C07331=1159.961,302.265,-72.493,-176.878,8.230,148.701
C07332=1159.957,302.514,-72.524,-176.876,8.233,148.700
C07333=1159.952,302.762,-72.555,-176.873,8.237,148.701
C07334=1159.948,303.010,-72.586,-176.871,8.239,148.701
C07335=1159.944,303.258,-72.616,-176.868,8.243,148.701
C07336=1159.940,303.506,-72.648,-176.866,8.246,148.701
C07337=1159.936,303.754,-72.679,-176.863,8.249,148.701
C07338=1159.932,304.002,-72.710,-176.861,8.252,148.701
C07339=1159.928,304.250,-72.740,-176.858,8.256,148.701
C07340=1159.923,304.498,-72.771,-176.855,8.259,148.701
C07341=1159.919,304.747,-72.802,-176.853,8.262,148.701
C07342=1159.914,304.994,-72.833,-176.850,8.265,148.701
C07343=1159.910,305.242,-72.863,-176.848,8.269,148.701
C07344=1159.906,305.490,-72.895,-176.845,8.272,148.701
C07345=1159.902,305.738,-72.925,-176.842,8.275,148.702
C07346=1159.898,305.986,-72.956,-176.840,8.278,148.702
C07347=1159.894,306.235,-72.987,-176.837,8.282,148.702
C07348=1159.889,306.482,-73.019,-176.835,8.285,148.702
C07349=1159.885,306.731,-73.050,-176.832,8.288,148.702
C07350=1159.881,306.979,-73.081,-176.830,8.291,148.702
C07351=1159.876,307.227,-73.111,-176.827,8.294,148.702
C07352=1159.873,307.474,-73.143,-176.824,8.298,148.702
C07353=1159.868,307.722,-73.173,-176.822,8.301,148.702
C07354=1159.864,307.971,-73.205,-176.819,8.305,148.703
C07355=1159.860,308.218,-73.236,-176.816,8.308,148.703
C07356=1159.856,308.466,-73.267,-176.814,8.311,148.703
C07357=1159.852,308.715,-73.298,-176.811,8.314,148.703
C07358=1159.847,308.962,-73.329,-176.809,8.317,148.703
C07359=1159.843,309.211,-73.361,-176.806,8.320,148.703
C07360=1159.839,309.458,-73.392,-176.804,8.323,148.703
C07361=1159.835,309.707,-73.423,-176.801,8.328,148.703
C07362=1159.830,309.955,-73.454,-176.798,8.331,148.703
C07363=1159.827,310.203,-73.486,-176.796,8.334,148.703
C07364=1159.822,310.451,-73.517,-176.793,8.337,148.704
C07365=1159.818,310.699,-73.548,-176.791,8.340,148.704
C07366=1159.814,310.947,-73.579,-176.788,8.343,148.704
C07367=1159.810,311.195,-73.611,-176.785,8.347,148.704
C07368=1159.805,311.443,-73.642,-176.783,8.350,148.704
C07369=1159.802,311.691,-73.674,-176.780,8.354,148.704
C07370=1159.797,311.939,-73.704,-176.778,8.357,148.704
C07371=1159.793,312.187,-73.736,-176.775,8.360,148.704
C07372=1159.789,312.434,-73.768,-176.773,8.363,148.705
C07373=1159.785,312.683,-73.799,-176.770,8.367,148.705
C07374=1159.781,312.930,-73.830,-176.767,8.370,148.705
C07375=1159.777,313.179,-73.861,-176.765,8.373,148.705
C07376=1159.772,313.456,-73.897,-176.762,8.377,148.705
C07377=1159.767,313.733,-73.932,-176.760,8.381,148.705
C07378=1159.762,314.010,-73.967,-176.756,8.384,148.705
C07379=1159.758,314.288,-74.003,-176.753,8.389,148.705
C07380=1159.754,314.536,-74.034,-176.751,8.392,148.705
C07381=1159.750,314.784,-74.066,-176.748,8.395,148.706
C07382=1159.745,315.031,-74.098,-176.746,8.398,148.706
C07383=1159.741,315.280,-74.129,-176.743,8.401,148.706
C07384=1159.737,315.528,-74.161,-176.741,8.404,148.706
C07385=1159.733,315.775,-74.192,-176.738,8.408,148.706
C07386=1159.729,316.023,-74.224,-176.735,8.411,148.706
C07387=1159.724,316.271,-74.256,-176.733,8.415,148.706
C07388=1159.720,316.520,-74.287,-176.731,8.418,148.707
C07389=1159.716,316.768,-74.319,-176.728,8.421,148.707
C07390=1159.712,317.015,-74.351,-176.725,8.425,148.707
C07391=1159.708,317.263,-74.382,-176.723,8.428,148.707
C07392=1159.703,317.511,-74.415,-176.720,8.431,148.707
C07393=1159.700,317.759,-74.446,-176.718,8.435,148.707
C07394=1159.696,318.007,-74.478,-176.715,8.438,148.707
C07395=1159.691,318.255,-74.509,-176.712,8.442,148.707
C07396=1159.687,318.503,-74.541,-176.710,8.445,148.708
C07397=1159.683,318.751,-74.573,-176.707,8.448,148.708
C07398=1159.679,318.998,-74.605,-176.705,8.451,148.708
C07399=1159.674,319.247,-74.637,-176.702,8.454,148.708
C07400=1159.671,319.495,-74.669,-176.699,8.459,148.708
C07401=1159.666,319.742,-74.701,-176.697,8.462,148.708
C07402=1159.663,319.990,-74.732,-176.694,8.465,148.708
C07403=1159.658,320.239,-74.765,-176.692,8.468,148.709
C07404=1159.654,320.487,-74.797,-176.689,8.472,148.709
C07405=1159.650,320.734,-74.828,-176.687,8.475,148.709
C07406=1159.646,320.982,-74.861,-176.684,8.478,148.709
C07407=1159.642,321.230,-74.892,-176.682,8.482,148.709
C07408=1159.637,321.478,-74.924,-176.680,8.485,148.709
C07409=1159.634,321.725,-74.957,-176.677,8.489,148.710
C07410=1159.630,321.973,-74.989,-176.674,8.492,148.710
C07411=1159.625,322.222,-75.021,-176.672,8.495,148.710
C07412=1159.621,322.469,-75.053,-176.669,8.499,148.710
C07413=1159.617,322.717,-75.085,-176.666,8.502,148.710
C07414=1159.613,322.966,-75.117,-176.664,8.506,148.710
C07415=1159.609,323.214,-75.149,-176.661,8.509,148.710
C07416=1159.604,323.461,-75.182,-176.659,8.512,148.711
C07417=1159.601,323.709,-75.214,-176.657,8.516,148.711
C07418=1159.596,323.957,-75.246,-176.653,8.519,148.711
C07419=1159.593,324.205,-75.278,-176.651,8.523,148.711
C07420=1159.588,324.453,-75.311,-176.649,8.526,148.711
C07421=1159.584,324.700,-75.342,-176.647,8.529,148.711
C07422=1159.580,324.948,-75.375,-176.643,8.533,148.711
C07423=1159.576,325.196,-75.407,-176.641,8.536,148.712
C07424=1159.572,325.444,-75.440,-176.639,8.540,148.712
C07425=1159.568,325.692,-75.472,-176.636,8.543,148.712
C07426=1159.563,325.940,-75.504,-176.633,8.547,148.712
C07427=1159.560,326.187,-75.536,-176.631,8.550,148.712
C07428=1159.555,326.436,-75.569,-176.628,8.553,148.712
C07429=1159.552,326.684,-75.601,-176.626,8.557,148.713
C07430=1159.547,326.931,-75.634,-176.623,8.561,148.713
C07431=1159.542,327.179,-75.666,-176.621,8.564,148.713
C07432=1159.539,327.426,-75.698,-176.618,8.567,148.713
C07433=1159.535,327.675,-75.731,-176.616,8.570,148.713
C07434=1159.531,327.922,-75.763,-176.613,8.574,148.713
C07435=1159.527,328.171,-75.796,-176.611,8.578,148.714
C07436=1159.522,328.419,-75.828,-176.608,8.581,148.714
C07437=1159.519,328.666,-75.861,-176.605,8.585,148.714
C07438=1159.514,328.914,-75.893,-176.603,8.588,148.714
C07439=1159.510,329.162,-75.926,-176.600,8.591,148.714
C07440=1159.506,329.409,-75.959,-176.598,8.594,148.715
C07441=1159.502,329.658,-75.991,-176.595,8.599,148.715
C07442=1159.498,329.905,-76.024,-176.593,8.602,148.715
C07443=1159.494,330.153,-76.056,-176.591,8.605,148.715
C07444=1159.490,330.401,-76.089,-176.588,8.608,148.715
C07445=1159.485,330.649,-76.122,-176.585,8.612,148.715
C07446=1159.482,330.897,-76.154,-176.583,8.615,148.716
C07447=1159.478,331.145,-76.187,-176.580,8.619,148.716
C07448=1159.473,331.393,-76.220,-176.578,8.623,148.716
C07449=1159.469,331.640,-76.253,-176.575,8.626,148.716
C07450=1159.465,331.887,-76.285,-176.573,8.629,148.716
C07451=1159.461,332.136,-76.318,-176.571,8.633,148.717
C07452=1159.457,332.383,-76.351,-176.567,8.637,148.717
C07453=1159.453,332.631,-76.384,-176.565,8.640,148.717
C07454=1159.448,332.879,-76.416,-176.563,8.643,148.717
C07455=1159.445,333.127,-76.449,-176.560,8.647,148.717
C07456=1159.441,333.375,-76.482,-176.557,8.650,148.718
C07457=1159.436,333.622,-76.515,-176.555,8.654,148.718
C07458=1159.432,333.871,-76.548,-176.553,8.657,148.718
C07459=1159.428,334.118,-76.581,-176.550,8.661,148.718
C07460=1159.424,334.366,-76.613,-176.548,8.664,148.718
C07461=1159.420,334.614,-76.647,-176.545,8.668,148.719
C07462=1159.416,334.861,-76.680,-176.543,8.672,148.719
C07463=1159.412,335.109,-76.713,-176.540,8.675,148.719
C07464=1159.408,335.357,-76.745,-176.537,8.678,148.719
C07465=1159.403,335.605,-76.779,-176.535,8.682,148.719
C07466=1159.399,335.853,-76.812,-176.532,8.685,148.719
C07467=1159.395,336.101,-76.845,-176.530,8.689,148.720
C07468=1159.392,336.348,-76.877,-176.527,8.693,148.720
C07469=1159.388,336.596,-76.911,-176.525,8.696,148.720
C07470=1159.384,336.843,-76.944,-176.522,8.699,148.720
C07471=1159.379,337.091,-76.977,-176.520,8.704,148.721
C07472=1159.375,337.339,-77.010,-176.517,8.707,148.721
C07473=1159.372,337.587,-77.044,-176.515,8.710,148.721
C07474=1159.368,337.835,-77.077,-176.512,8.714,148.721
C07475=1159.363,338.083,-77.110,-176.510,8.717,148.721
C07476=1159.359,338.331,-77.143,-176.507,8.721,148.722
C07477=1159.355,338.578,-77.176,-176.505,8.725,148.722
C07478=1159.351,338.826,-77.209,-176.502,8.728,148.722
C07479=1159.347,339.074,-77.243,-176.500,8.731,148.722
C07480=1159.342,339.353,-77.280,-176.497,8.736,148.723
C07481=1159.338,339.633,-77.318,-176.494,8.740,148.723
C07482=1159.334,339.913,-77.355,-176.491,8.744,148.723
C07483=1159.329,340.193,-77.393,-176.488,8.748,148.723
C07484=1159.324,340.441,-77.427,-176.486,8.751,148.724
C07485=1159.320,340.689,-77.460,-176.483,8.755,148.724
C07486=1159.316,340.936,-77.493,-176.481,8.759,148.724
C07487=1159.312,341.183,-77.527,-176.479,8.762,148.724
C07488=1159.308,341.431,-77.560,-176.476,8.766,148.724
C07489=1159.304,341.679,-77.593,-176.473,8.769,148.725
C07490=1159.300,341.927,-77.627,-176.471,8.772,148.725
C07491=1159.296,342.174,-77.661,-176.468,8.777,148.725
C07492=1159.292,342.422,-77.694,-176.466,8.780,148.725
C07493=1159.287,342.670,-77.728,-176.464,8.783,148.726
C07494=1159.283,342.918,-77.761,-176.461,8.787,148.726
C07495=1159.279,343.165,-77.795,-176.458,8.791,148.726
C07496=1159.276,343.413,-77.828,-176.456,8.794,148.726
C07497=1159.272,343.661,-77.861,-176.453,8.798,148.726
C07498=1159.268,343.908,-77.895,-176.451,8.801,148.727
C07499=1159.263,344.156,-77.929,-176.449,8.806,148.727
C07500=1159.259,344.404,-77.962,-176.446,8.809,148.727
C07501=1159.256,344.652,-77.996,-176.444,8.812,148.728
C07502=1159.252,344.900,-78.029,-176.441,8.816,148.728
C07503=1159.247,345.147,-78.064,-176.439,8.820,148.728
C07504=1159.243,345.395,-78.097,-176.436,8.823,148.728
C07505=1159.239,345.642,-78.131,-176.434,8.827,148.728
C07506=1159.236,345.890,-78.164,-176.431,8.830,148.729
C07507=1159.231,346.138,-78.199,-176.428,8.834,148.729
C07508=1159.227,346.385,-78.232,-176.426,8.838,148.729
C07509=1159.223,346.632,-78.266,-176.424,8.841,148.729
C07510=1159.219,346.881,-78.299,-176.421,8.845,148.730
C07511=1159.215,347.128,-78.334,-176.419,8.849,148.730
C07512=1159.211,347.376,-78.367,-176.416,8.853,148.730
C07513=1159.208,347.624,-78.401,-176.414,8.856,148.730
C07514=1159.203,347.872,-78.435,-176.411,8.859,148.731
C07515=1159.199,348.119,-78.469,-176.409,8.863,148.731
C07516=1159.195,348.366,-78.503,-176.406,8.867,148.731
C07517=1159.191,348.615,-78.537,-176.404,8.871,148.732
C07518=1159.187,348.862,-78.571,-176.402,8.874,148.732
C07519=1159.183,349.110,-78.604,-176.399,8.878,148.732
C07520=1159.179,349.358,-78.639,-176.396,8.882,148.732
C07521=1159.175,349.605,-78.673,-176.394,8.885,148.733
C07522=1159.170,349.853,-78.706,-176.391,8.889,148.733
C07523=1159.167,350.101,-78.741,-176.389,8.892,148.733
C07524=1159.163,350.348,-78.775,-176.386,8.897,148.733
C07525=1159.158,350.595,-78.809,-176.384,8.900,148.734
C07526=1159.155,350.844,-78.843,-176.382,8.903,148.734
C07527=1159.150,351.091,-78.877,-176.379,8.908,148.734
C07528=1159.146,351.338,-78.911,-176.377,8.911,148.734
C07529=1159.143,351.586,-78.946,-176.374,8.915,148.735
C07530=1159.139,351.834,-78.980,-176.372,8.919,148.735
C07531=1159.134,352.082,-79.013,-176.369,8.923,148.735
C07532=1159.131,352.329,-79.048,-176.367,8.926,148.736
C07533=1159.126,352.577,-79.082,-176.364,8.929,148.736
C07534=1159.123,352.825,-79.116,-176.362,8.934,148.736
C07535=1159.118,353.072,-79.151,-176.360,8.937,148.736
C07536=1159.114,353.319,-79.185,-176.357,8.941,148.737
C07537=1159.110,353.567,-79.219,-176.354,8.944,148.737
C07538=1159.107,353.814,-79.253,-176.352,8.949,148.737
C07539=1159.103,354.062,-79.288,-176.350,8.952,148.738
C07540=1159.099,354.310,-79.322,-176.347,8.956,148.738
C07541=1159.094,354.557,-79.356,-176.344,8.959,148.738
C07542=1159.091,354.805,-79.390,-176.343,8.963,148.738
C07543=1159.086,355.053,-79.424,-176.340,8.967,148.739
C07544=1159.083,355.300,-79.459,-176.337,8.970,148.739
C07545=1159.079,355.547,-79.494,-176.335,8.974,148.739
C07546=1159.075,355.796,-79.529,-176.333,8.978,148.740
C07547=1159.071,356.043,-79.563,-176.330,8.982,148.740
C07548=1159.067,356.291,-79.597,-176.327,8.985,148.740
C07549=1159.062,356.538,-79.632,-176.325,8.990,148.741
C07550=1159.059,356.786,-79.666,-176.323,8.993,148.741
C07551=1159.054,357.033,-79.701,-176.320,8.997,148.741
C07552=1159.051,357.281,-79.735,-176.317,9.001,148.741
C07553=1159.047,357.529,-79.769,-176.315,9.005,148.742
C07554=1159.043,357.777,-79.804,-176.313,9.008,148.742
C07555=1159.039,358.023,-79.839,-176.310,9.012,148.742
C07556=1159.035,358.271,-79.874,-176.308,9.016,148.743
C07557=1159.031,358.519,-79.908,-176.305,9.020,148.743
C07558=1159.027,358.767,-79.943,-176.303,9.023,148.743
C07559=1159.023,359.013,-79.977,-176.300,9.028,148.744
C07560=1159.019,359.262,-80.012,-176.298,9.031,148.744
C07561=1159.015,359.509,-80.047,-176.295,9.035,148.744
C07562=1159.011,359.757,-80.081,-176.293,9.039,148.744
C07563=1159.007,360.004,-80.116,-176.290,9.043,148.745
C07564=1159.003,360.252,-80.151,-176.288,9.046,148.745
C07565=1158.999,360.499,-80.185,-176.286,9.051,148.745
C07566=1158.996,360.746,-80.220,-176.283,9.054,148.746
C07567=1158.992,360.994,-80.255,-176.280,9.058,148.746
C07568=1158.987,361.242,-80.290,-176.279,9.062,148.746
C07569=1158.983,361.489,-80.325,-176.276,9.066,148.747
C07570=1158.979,361.737,-80.360,-176.273,9.070,148.747
C07571=1158.976,361.985,-80.394,-176.271,9.073,148.747
C07572=1158.972,362.232,-80.429,-176.268,9.077,148.748
C07573=1158.967,362.480,-80.464,-176.266,9.081,148.748
C07574=1158.964,362.727,-80.499,-176.263,9.085,148.748
C07575=1158.959,362.974,-80.534,-176.261,9.089,148.749
C07576=1158.955,363.222,-80.569,-176.258,9.093,148.749
C07577=1158.952,363.470,-80.604,-176.256,9.097,148.749
C07578=1158.948,363.717,-80.639,-176.254,9.101,148.750
C07579=1158.944,363.965,-80.674,-176.251,9.105,148.750
C07580=1158.940,364.212,-80.709,-176.249,9.108,148.750
C07581=1158.936,364.460,-80.744,-176.246,9.112,148.751
C07582=1158.932,364.707,-80.779,-176.244,9.116,148.751
C07583=1158.928,364.955,-80.815,-176.241,9.120,148.751
C07584=1158.924,365.238,-80.854,-176.239,9.124,148.752
C07585=1158.919,365.520,-80.894,-176.236,9.129,148.752
C07586=1158.915,365.803,-80.934,-176.234,9.133,148.752
C07587=1158.910,366.086,-80.975,-176.230,9.138,148.753
C07588=1158.906,366.333,-81.010,-176.229,9.142,148.753
C07589=1158.902,366.580,-81.046,-176.226,9.146,148.754
C07590=1158.898,366.828,-81.081,-176.224,9.149,148.754
C07591=1158.894,367.075,-81.116,-176.221,9.154,148.755
C07592=1158.890,367.323,-81.151,-176.220,9.157,148.755
C07593=1158.886,367.571,-81.186,-176.217,9.162,148.755
C07594=1158.883,367.818,-81.222,-176.215,9.165,148.756
C07595=1158.878,368.065,-81.257,-176.212,9.170,148.756
C07596=1158.875,368.313,-81.292,-176.210,9.173,148.757
C07597=1158.871,368.560,-81.328,-176.208,9.177,148.757
C07598=1158.867,368.808,-81.362,-176.206,9.181,148.757
C07599=1158.863,369.055,-81.398,-176.203,9.185,148.758
C07600=1158.859,369.303,-81.433,-176.201,9.189,148.758
C07601=1158.856,369.550,-81.469,-176.199,9.193,148.759
C07602=1158.851,369.797,-81.504,-176.197,9.197,148.759
C07603=1158.848,370.044,-81.540,-176.195,9.201,148.760
C07604=1158.843,370.292,-81.576,-176.193,9.205,148.760
C07605=1158.839,370.540,-81.611,-176.191,9.208,148.760
C07606=1158.836,370.788,-81.646,-176.188,9.213,148.761
C07607=1158.831,371.035,-81.681,-176.186,9.216,148.761
C07608=1158.828,371.282,-81.717,-176.184,9.221,148.762
C07609=1158.824,371.530,-81.753,-176.182,9.224,148.762
C07610=1158.820,371.777,-81.788,-176.180,9.228,148.763
C07611=1158.816,372.025,-81.824,-176.178,9.233,148.763
C07612=1158.812,372.272,-81.859,-176.176,9.236,148.764
C07613=1158.808,372.519,-81.895,-176.174,9.241,148.764
C07614=1158.804,372.767,-81.931,-176.172,9.244,148.765
C07615=1158.801,373.014,-81.966,-176.171,9.248,148.765
C07616=1158.796,373.262,-82.002,-176.169,9.252,148.766
C07617=1158.793,373.509,-82.038,-176.166,9.256,148.766
C07618=1158.788,373.756,-82.073,-176.165,9.260,148.767
C07619=1158.785,374.003,-82.109,-176.163,9.264,148.767
C07620=1158.781,374.251,-82.145,-176.161,9.268,148.768
C07621=1158.777,374.498,-82.181,-176.159,9.272,148.768
C07622=1158.773,374.746,-82.216,-176.158,9.276,148.769
C07623=1158.770,374.993,-82.252,-176.156,9.280,148.769
C07624=1158.765,375.241,-82.288,-176.154,9.283,148.770
C07625=1158.761,375.488,-82.323,-176.153,9.287,148.771
C07626=1158.758,375.735,-82.360,-176.150,9.292,148.771
C07627=1158.753,375.983,-82.396,-176.149,9.296,148.772
C07628=1158.750,376.230,-82.431,-176.147,9.300,148.772
C07629=1158.746,376.478,-82.467,-176.146,9.303,148.773
C07630=1158.742,376.725,-82.502,-176.144,9.307,148.774
C07631=1158.738,376.972,-82.539,-176.143,9.311,148.774
C07632=1158.734,377.220,-82.575,-176.141,9.315,148.775
C07633=1158.731,377.467,-82.610,-176.140,9.319,148.775
C07634=1158.726,377.715,-82.646,-176.138,9.323,148.776
C07635=1158.722,377.961,-82.682,-176.137,9.327,148.776
C07636=1158.718,378.209,-82.719,-176.135,9.330,148.777
C07637=1158.714,378.457,-82.754,-176.134,9.334,148.778
C07638=1158.711,378.704,-82.790,-176.133,9.339,148.779
C07639=1158.707,378.951,-82.826,-176.131,9.342,148.779
C07640=1158.703,379.199,-82.862,-176.131,9.346,148.780
C07641=1158.699,379.446,-82.899,-176.129,9.349,148.780
C07642=1158.695,379.694,-82.934,-176.128,9.354,148.781
C07643=1158.692,379.941,-82.970,-176.127,9.358,148.782
C07644=1158.687,380.188,-83.007,-176.126,9.361,148.782
C07645=1158.684,380.436,-83.042,-176.125,9.365,148.783
C07646=1158.680,380.683,-83.079,-176.123,9.369,148.784
C07647=1158.676,380.931,-83.115,-176.123,9.372,148.785
C07648=1158.672,381.178,-83.151,-176.121,9.376,148.785
C07649=1158.668,381.425,-83.187,-176.120,9.380,148.786
C07650=1158.665,381.673,-83.223,-176.119,9.383,148.787
C07651=1158.661,381.920,-83.260,-176.118,9.388,148.787
C07652=1158.656,382.167,-83.295,-176.118,9.391,148.788
C07653=1158.652,382.414,-83.332,-176.117,9.395,148.789
C07654=1158.649,382.661,-83.367,-176.116,9.398,148.790
C07655=1158.644,382.909,-83.404,-176.116,9.402,148.790
C07656=1158.641,383.156,-83.440,-176.114,9.405,148.791
C07657=1158.637,383.403,-83.476,-176.114,9.409,148.792
C07658=1158.633,383.651,-83.512,-176.113,9.412,148.793
C07659=1158.629,383.898,-83.549,-176.112,9.416,148.793
C07660=1158.625,384.145,-83.584,-176.112,9.420,148.794
C07661=1158.621,384.393,-83.621,-176.111,9.423,148.795
C07662=1158.617,384.640,-83.657,-176.111,9.427,148.796
C07663=1158.613,384.887,-83.694,-176.110,9.430,148.796
C07664=1158.610,385.136,-83.730,-176.110,9.433,148.797
C07665=1158.606,385.383,-83.766,-176.110,9.437,148.798
C07666=1158.602,385.630,-83.803,-176.109,9.440,148.799
C07667=1158.598,385.877,-83.839,-176.109,9.444,148.800
C07668=1158.594,386.125,-83.876,-176.109,9.447,148.800
C07669=1158.591,386.372,-83.911,-176.109,9.450,148.801
C07670=1158.587,386.619,-83.948,-176.108,9.453,148.802
C07671=1158.583,386.866,-83.984,-176.108,9.457,148.803
C07672=1158.579,387.114,-84.021,-176.108,9.460,148.804
C07673=1158.576,387.361,-84.057,-176.108,9.463,148.804
C07674=1158.571,387.608,-84.094,-176.108,9.467,148.805
C07675=1158.567,387.856,-84.130,-176.108,9.469,148.806
C07676=1158.564,388.103,-84.166,-176.108,9.472,148.807
C07677=1158.560,388.350,-84.203,-176.108,9.475,148.808
C07678=1158.556,388.597,-84.238,-176.108,9.479,148.808
C07679=1158.552,388.845,-84.275,-176.108,9.482,148.809
C07680=1158.548,389.092,-84.312,-176.108,9.484,148.810
C07681=1158.544,389.339,-84.348,-176.108,9.488,148.811
C07682=1158.540,389.587,-84.385,-176.109,9.490,148.812
C07683=1158.537,389.833,-84.421,-176.109,9.493,148.813
C07684=1158.532,390.081,-84.457,-176.109,9.497,148.813
C07685=1158.529,390.328,-84.493,-176.109,9.500,148.814
C07686=1158.525,390.576,-84.530,-176.109,9.502,148.815
C07687=1158.521,390.824,-84.567,-176.110,9.505,148.816
C07688=1158.517,391.109,-84.609,-176.110,9.508,148.817
C07689=1158.512,391.395,-84.651,-176.110,9.512,148.818
C07690=1158.508,391.680,-84.693,-176.111,9.514,148.819
C07691=1158.503,391.966,-84.735,-176.112,9.517,148.820
C07692=1158.500,392.214,-84.772,-176.112,9.520,148.820
C07693=1158.496,392.461,-84.808,-176.112,9.523,148.821
C07694=1158.492,392.709,-84.844,-176.113,9.526,148.822
C07695=1158.488,392.956,-84.881,-176.113,9.529,148.823
C07696=1158.484,393.203,-84.918,-176.113,9.531,148.824
C07697=1158.480,393.451,-84.954,-176.114,9.534,148.825
C07698=1158.477,393.698,-84.990,-176.115,9.536,148.825
C07699=1158.472,393.945,-85.027,-176.115,9.539,148.826
C07700=1158.468,394.192,-85.064,-176.116,9.541,148.827
C07701=1158.465,394.439,-85.099,-176.116,9.543,148.828
C07702=1158.461,394.687,-85.136,-176.117,9.546,148.829
C07703=1158.457,394.934,-85.173,-176.117,9.549,148.829
C07704=1158.454,395.181,-85.210,-176.118,9.551,148.830
C07705=1158.450,395.429,-85.246,-176.119,9.554,148.831
C07706=1158.445,395.676,-85.283,-176.119,9.556,148.832
C07707=1158.442,395.923,-85.319,-176.120,9.558,148.833
C07708=1158.438,396.170,-85.356,-176.120,9.561,148.833
C07709=1158.434,396.418,-85.393,-176.121,9.563,148.834
C07710=1158.430,396.665,-85.428,-176.122,9.566,148.835
C07711=1158.426,396.912,-85.465,-176.123,9.567,148.836
C07712=1158.422,397.159,-85.502,-176.123,9.570,148.837
C07713=1158.419,397.406,-85.538,-176.124,9.572,148.837
C07714=1158.414,397.654,-85.575,-176.124,9.575,148.838
C07715=1158.410,397.901,-85.611,-176.125,9.577,148.839
C07716=1158.407,398.149,-85.648,-176.126,9.579,148.840
C07717=1158.403,398.396,-85.685,-176.126,9.581,148.840
C07718=1158.399,398.643,-85.721,-176.127,9.583,148.841
C07719=1158.395,398.891,-85.757,-176.128,9.586,148.842
C07720=1158.391,399.138,-85.794,-176.129,9.588,148.843
C07721=1158.387,399.385,-85.831,-176.129,9.590,148.843
C07722=1158.384,399.632,-85.867,-176.131,9.592,148.844
C07723=1158.380,399.879,-85.904,-176.131,9.594,148.845
C07724=1158.375,400.127,-85.940,-176.132,9.596,148.846
C07725=1158.372,400.374,-85.976,-176.132,9.598,148.846
C07726=1158.369,400.622,-86.013,-176.133,9.601,148.847
C07727=1158.364,400.869,-86.050,-176.134,9.603,148.848
C07728=1158.361,401.116,-86.087,-176.134,9.605,148.849
C07729=1158.357,401.364,-86.123,-176.136,9.607,148.849
C07730=1158.353,401.611,-86.160,-176.136,9.608,148.850
C07731=1158.349,401.858,-86.196,-176.137,9.611,148.851
C07732=1158.345,402.105,-86.233,-176.137,9.613,148.852
C07733=1158.341,402.352,-86.270,-176.138,9.615,148.852
C07734=1158.337,402.599,-86.306,-176.139,9.617,148.853
C07735=1158.333,402.847,-86.342,-176.140,9.619,148.854
C07736=1158.330,403.095,-86.379,-176.140,9.621,148.854
C07737=1158.326,403.342,-86.416,-176.141,9.623,148.855
C07738=1158.322,403.589,-86.452,-176.142,9.625,148.856
C07739=1158.318,403.836,-86.489,-176.143,9.627,148.857
C07740=1158.314,404.084,-86.525,-176.143,9.628,148.857
C07741=1158.310,404.331,-86.562,-176.144,9.630,148.858
C07742=1158.306,404.578,-86.598,-176.145,9.632,148.859
C07743=1158.302,404.825,-86.635,-176.145,9.635,148.859
C07744=1158.299,405.072,-86.672,-176.146,9.637,148.860
C07745=1158.295,405.320,-86.709,-176.147,9.639,148.861
C07746=1158.291,405.568,-86.745,-176.148,9.640,148.862
C07747=1158.287,405.815,-86.782,-176.148,9.642,148.862
C07748=1158.284,406.062,-86.818,-176.149,9.644,148.863
C07749=1158.279,406.309,-86.855,-176.150,9.646,148.864
C07750=1158.275,406.556,-86.892,-176.151,9.647,148.864
C07751=1158.272,406.803,-86.928,-176.151,9.649,148.865
C07752=1158.268,407.050,-86.965,-176.152,9.651,148.866
C07753=1158.264,407.298,-87.001,-176.152,9.654,148.866
C07754=1158.261,407.546,-87.038,-176.153,9.655,148.867
C07755=1158.257,407.793,-87.075,-176.154,9.657,148.868
C07756=1158.253,408.040,-87.111,-176.155,9.659,148.868
C07757=1158.248,408.287,-87.148,-176.155,9.661,148.869
C07758=1158.245,408.534,-87.184,-176.156,9.662,148.870
C07759=1158.241,408.782,-87.221,-176.157,9.664,148.870
C07760=1158.237,409.029,-87.257,-176.157,9.666,148.871
C07761=1158.233,409.276,-87.294,-176.158,9.668,148.872
C07762=1158.229,409.523,-87.331,-176.159,9.669,148.872
C07763=1158.226,409.771,-87.368,-176.159,9.671,148.873
C07764=1158.222,410.018,-87.404,-176.160,9.673,148.873
C07765=1158.218,410.265,-87.441,-176.160,9.675,148.874
C07766=1158.214,410.513,-87.477,-176.161,9.677,148.875
C07767=1158.210,410.760,-87.514,-176.162,9.679,148.875
C07768=1158.206,411.007,-87.550,-176.162,9.681,148.876
C07769=1158.202,411.254,-87.587,-176.163,9.682,148.877
C07770=1158.198,411.501,-87.624,-176.164,9.684,148.877
C07771=1158.195,411.749,-87.661,-176.164,9.686,148.878
C07772=1158.191,411.996,-87.697,-176.165,9.687,148.879
C07773=1158.187,412.244,-87.734,-176.165,9.689,148.879
C07774=1158.183,412.491,-87.770,-176.166,9.691,148.880
C07775=1158.180,412.738,-87.807,-176.167,9.693,148.880
C07776=1158.175,412.985,-87.844,-176.167,9.695,148.881
C07777=1158.171,413.232,-87.880,-176.168,9.697,148.882
C07778=1158.167,413.480,-87.917,-176.168,9.698,148.882
C07779=1158.164,413.727,-87.954,-176.168,9.700,148.883
C07780=1158.160,413.974,-87.991,-176.169,9.702,148.884
C07781=1158.156,414.222,-88.027,-176.170,9.704,148.884
C07782=1158.153,414.469,-88.063,-176.171,9.705,148.885
C07783=1158.149,414.716,-88.100,-176.171,9.707,148.885
C07784=1158.144,414.963,-88.137,-176.171,9.709,148.886
C07785=1158.142,415.211,-88.173,-176.172,9.711,148.887
C07786=1158.138,415.458,-88.210,-176.172,9.713,148.887
C07787=1158.137,415.705,-88.247,-176.173,9.714,148.888
C07788=1158.136,416.085,-88.302,-176.173,9.717,148.889
C07789=1158.136,416.464,-88.358,-176.174,9.719,148.889
C07790=1158.140,416.843,-88.413,-176.175,9.722,148.890
C07791=1158.145,417.220,-88.468,-176.175,9.725,148.891
C07792=1157.724,417.222,-88.515,-176.178,9.736,148.895
C07793=1157.719,416.841,-88.460,-176.178,9.733,148.894
C07794=1157.716,416.459,-88.404,-176.177,9.731,148.893
C07795=1157.716,416.076,-88.348,-176.176,9.728,148.892
C07796=1157.716,415.693,-88.292,-176.176,9.725,148.891
C07797=1157.718,415.447,-88.255,-176.175,9.724,148.891
C07798=1157.720,415.200,-88.219,-176.174,9.722,148.890
C07799=1157.724,414.952,-88.182,-176.174,9.720,148.890
C07800=1157.727,414.705,-88.145,-176.173,9.719,148.889
C07801=1157.731,414.458,-88.109,-176.173,9.716,148.888
C07802=1157.736,414.210,-88.072,-176.173,9.714,148.888
C07803=1157.740,413.963,-88.036,-176.172,9.713,148.887
C07804=1157.743,413.716,-87.999,-176.172,9.711,148.887
C07805=1157.747,413.469,-87.962,-176.171,9.709,148.886
C07806=1157.751,413.221,-87.926,-176.170,9.708,148.885
C07807=1157.755,412.973,-87.888,-176.170,9.706,148.885
C07808=1157.758,412.727,-87.852,-176.169,9.704,148.884
C07809=1157.762,412.479,-87.815,-176.168,9.702,148.883
C07810=1157.766,412.232,-87.778,-176.168,9.700,148.883
C07811=1157.771,411.984,-87.742,-176.167,9.698,148.882
C07812=1157.774,411.738,-87.706,-176.167,9.697,148.882
C07813=1157.778,411.490,-87.669,-176.166,9.695,148.881
C07814=1157.782,411.243,-87.632,-176.166,9.693,148.880
C07815=1157.785,410.996,-87.596,-176.165,9.691,148.880
C07816=1157.789,410.748,-87.559,-176.164,9.690,148.879
C07817=1157.793,410.501,-87.522,-176.164,9.688,148.878
C07818=1157.797,410.254,-87.485,-176.163,9.686,148.878
C07819=1157.801,410.006,-87.450,-176.162,9.684,148.877
C07820=1157.805,409.759,-87.413,-176.162,9.683,148.876
C07821=1157.809,409.512,-87.376,-176.161,9.680,148.876
C07822=1157.812,409.265,-87.340,-176.161,9.678,148.875
C07823=1157.816,409.017,-87.302,-176.160,9.677,148.874
C07824=1157.820,408.770,-87.265,-176.159,9.675,148.874
C07825=1157.824,408.523,-87.229,-176.159,9.673,148.873
C07826=1157.828,408.275,-87.193,-176.158,9.671,148.873
C07827=1157.832,408.028,-87.156,-176.157,9.670,148.872
C07828=1157.836,407.781,-87.119,-176.157,9.668,148.871
C07829=1157.839,407.534,-87.083,-176.156,9.666,148.871
C07830=1157.843,407.287,-87.046,-176.155,9.664,148.870
C07831=1157.847,407.040,-87.009,-176.154,9.662,148.869
C07832=1157.851,406.792,-86.972,-176.153,9.661,148.868
C07833=1157.855,406.544,-86.937,-176.153,9.659,148.868
C07834=1157.859,406.297,-86.900,-176.153,9.656,148.867
C07835=1157.863,406.050,-86.863,-176.152,9.655,148.866
C07836=1157.866,405.803,-86.827,-176.151,9.653,148.866
C07837=1157.870,405.556,-86.790,-176.150,9.651,148.865
C07838=1157.874,405.309,-86.753,-176.149,9.649,148.864
C07839=1157.878,405.062,-86.717,-176.149,9.647,148.864
C07840=1157.882,404.813,-86.680,-176.148,9.645,148.863
C07841=1157.886,404.566,-86.643,-176.147,9.643,148.862
C07842=1157.890,404.319,-86.606,-176.146,9.642,148.862
C07843=1157.893,404.072,-86.570,-176.145,9.640,148.861
C07844=1157.897,403.825,-86.533,-176.145,9.637,148.860
C07845=1157.901,403.578,-86.496,-176.144,9.635,148.859
C07846=1157.905,403.330,-86.461,-176.144,9.634,148.859
C07847=1157.909,403.083,-86.424,-176.143,9.632,148.858
C07848=1157.913,402.836,-86.387,-176.142,9.630,148.857
C07849=1157.916,402.588,-86.351,-176.141,9.628,148.857
C07850=1157.920,402.341,-86.314,-176.140,9.626,148.856
C07851=1157.924,402.094,-86.277,-176.140,9.623,148.855
C07852=1157.928,401.846,-86.241,-176.139,9.622,148.854
C07853=1157.932,401.599,-86.204,-176.138,9.620,148.854
C07854=1157.936,401.352,-86.168,-176.137,9.618,148.853
C07855=1157.940,401.105,-86.131,-176.137,9.616,148.852
C07856=1157.943,400.858,-86.094,-176.136,9.613,148.851
C07857=1157.947,400.611,-86.058,-176.135,9.611,148.851
C07858=1157.952,400.363,-86.021,-176.134,9.609,148.850
C07859=1157.955,400.115,-85.985,-176.134,9.608,148.849
C07860=1157.959,399.868,-85.948,-176.133,9.605,148.848
C07861=1157.963,399.621,-85.911,-176.132,9.603,148.848
C07862=1157.966,399.374,-85.875,-176.132,9.601,148.847
C07863=1157.971,399.126,-85.839,-176.130,9.599,148.846
C07864=1157.975,398.879,-85.802,-176.130,9.597,148.845
C07865=1157.979,398.632,-85.765,-176.129,9.595,148.845
C07866=1157.982,398.385,-85.729,-176.128,9.592,148.844
C07867=1157.986,398.138,-85.692,-176.128,9.590,148.843
C07868=1157.990,397.890,-85.655,-176.127,9.588,148.842
C07869=1157.993,397.642,-85.619,-176.127,9.585,148.841
C07870=1157.997,397.395,-85.582,-176.126,9.583,148.841
C07871=1158.002,397.148,-85.545,-176.125,9.582,148.840
C07872=1158.005,396.901,-85.509,-176.124,9.579,148.839
C07873=1158.009,396.653,-85.473,-176.124,9.577,148.838
C07874=1158.013,396.406,-85.436,-176.123,9.574,148.838
C07875=1158.017,396.159,-85.400,-176.122,9.572,148.837
C07876=1158.021,395.912,-85.363,-176.122,9.569,148.836
C07877=1158.025,395.665,-85.326,-176.121,9.567,148.835
C07878=1158.029,395.417,-85.291,-176.121,9.565,148.834
C07879=1158.032,395.170,-85.253,-176.120,9.562,148.834
C07880=1158.036,394.922,-85.216,-176.119,9.560,148.833
C07881=1158.040,394.675,-85.180,-176.119,9.557,148.832
C07882=1158.044,394.428,-85.143,-176.118,9.554,148.831
C07883=1158.048,394.180,-85.107,-176.117,9.552,148.830
C07884=1158.051,393.934,-85.071,-176.117,9.550,148.830
C07885=1158.055,393.686,-85.034,-176.116,9.547,148.829
C07886=1158.060,393.439,-84.997,-176.116,9.545,148.828
C07887=1158.063,393.192,-84.962,-176.115,9.542,148.827
C07888=1158.067,392.945,-84.925,-176.115,9.539,148.826
C07889=1158.071,392.698,-84.889,-176.115,9.537,148.825
C07890=1158.075,392.450,-84.852,-176.114,9.534,148.825
C07891=1158.079,392.202,-84.815,-176.113,9.531,148.824
C07892=1158.082,391.955,-84.779,-176.113,9.529,148.823
C07893=1158.087,391.670,-84.736,-176.113,9.526,148.822
C07894=1158.092,391.384,-84.694,-176.112,9.523,148.821
C07895=1158.096,391.098,-84.653,-176.111,9.520,148.820
C07896=1158.100,390.812,-84.610,-176.111,9.516,148.819
C07897=1158.103,390.565,-84.574,-176.111,9.513,148.818
C07898=1158.108,390.317,-84.537,-176.111,9.510,148.817
C07899=1158.112,390.070,-84.501,-176.110,9.508,148.817
C07900=1158.115,389.823,-84.464,-176.110,9.505,148.816
C07901=1158.120,389.575,-84.428,-176.110,9.502,148.815
C07902=1158.123,389.328,-84.392,-176.110,9.499,148.814
C07903=1158.127,389.081,-84.355,-176.110,9.496,148.813
C07904=1158.131,388.833,-84.319,-176.110,9.492,148.813
C07905=1158.135,388.586,-84.283,-176.110,9.490,148.812
C07906=1158.139,388.339,-84.246,-176.109,9.487,148.811
C07907=1158.143,388.092,-84.210,-176.109,9.484,148.810
C07908=1158.147,387.844,-84.173,-176.109,9.481,148.809
C07909=1158.150,387.597,-84.136,-176.109,9.477,148.808
C07910=1158.154,387.349,-84.101,-176.109,9.475,148.808
C07911=1158.158,387.102,-84.064,-176.109,9.471,148.807
C07912=1158.161,386.855,-84.027,-176.110,9.468,148.806
C07913=1158.166,386.607,-83.991,-176.110,9.465,148.805
C07914=1158.169,386.360,-83.955,-176.110,9.461,148.804
C07915=1158.173,386.113,-83.918,-176.110,9.458,148.804
C07916=1158.178,385.865,-83.882,-176.111,9.455,148.803
C07917=1158.181,385.618,-83.846,-176.111,9.451,148.802
C07918=1158.185,385.371,-83.810,-176.111,9.448,148.801
C07919=1158.189,385.124,-83.773,-176.111,9.444,148.800
C07920=1158.193,384.877,-83.736,-176.112,9.441,148.800
C07921=1158.196,384.629,-83.701,-176.112,9.437,148.799
C07922=1158.200,384.382,-83.664,-176.113,9.434,148.798
C07923=1158.204,384.134,-83.629,-176.113,9.431,148.797
C07924=1158.208,383.887,-83.592,-176.114,9.427,148.797
C07925=1158.212,383.640,-83.556,-176.114,9.424,148.796
C07926=1158.216,383.392,-83.519,-176.116,9.420,148.795
C07927=1158.220,383.145,-83.484,-176.116,9.417,148.794
C07928=1158.224,382.898,-83.447,-176.116,9.413,148.794
C07929=1158.227,382.651,-83.411,-176.118,9.409,148.793
C07930=1158.232,382.403,-83.374,-176.118,9.406,148.792
C07931=1158.235,382.156,-83.338,-176.119,9.402,148.791
C07932=1158.239,381.908,-83.302,-176.120,9.398,148.791
C07933=1158.243,381.661,-83.267,-176.121,9.394,148.790
C07934=1158.247,381.414,-83.230,-176.122,9.391,148.789
C07935=1158.251,381.166,-83.194,-176.123,9.387,148.788
C07936=1158.255,380.919,-83.157,-176.124,9.384,148.788
C07937=1158.258,380.672,-83.122,-176.125,9.380,148.787
C07938=1158.263,380.424,-83.085,-176.126,9.376,148.786
C07939=1158.266,380.177,-83.049,-176.127,9.372,148.786
C07940=1158.270,379.930,-83.013,-176.128,9.368,148.785
C07941=1158.274,379.682,-82.977,-176.129,9.365,148.784
C07942=1158.278,379.435,-82.941,-176.131,9.360,148.784
C07943=1158.282,379.187,-82.904,-176.131,9.357,148.783
C07944=1158.285,378.940,-82.869,-176.133,9.353,148.782
C07945=1158.290,378.693,-82.833,-176.134,9.349,148.782
C07946=1158.294,378.446,-82.797,-176.136,9.346,148.781
C07947=1158.297,378.198,-82.761,-176.137,9.342,148.781
C07948=1158.302,377.951,-82.725,-176.139,9.338,148.780
C07949=1158.305,377.704,-82.689,-176.140,9.334,148.779
C07950=1158.309,377.456,-82.653,-176.142,9.330,148.779
C07951=1158.313,377.208,-82.617,-176.143,9.326,148.778
C07952=1158.317,376.961,-82.582,-176.144,9.322,148.777
C07953=1158.321,376.714,-82.545,-176.146,9.318,148.777
C07954=1158.325,376.466,-82.509,-176.147,9.314,148.776
C07955=1158.328,376.219,-82.474,-176.149,9.310,148.776
C07956=1158.333,375.972,-82.439,-176.151,9.307,148.775
C07957=1158.337,375.725,-82.402,-176.152,9.303,148.775
C07958=1158.340,375.477,-82.366,-176.154,9.298,148.774
C07959=1158.344,375.230,-82.331,-176.156,9.295,148.773
C07960=1158.348,374.982,-82.294,-176.158,9.291,148.773
C07961=1158.352,374.734,-82.259,-176.159,9.287,148.772
C07962=1158.356,374.487,-82.223,-176.161,9.283,148.772
C07963=1158.359,374.240,-82.187,-176.163,9.279,148.771
C07964=1158.364,373.993,-82.151,-176.165,9.275,148.771
C07965=1158.368,373.745,-82.116,-176.166,9.271,148.770
C07966=1158.371,373.498,-82.080,-176.169,9.267,148.770
C07967=1158.375,373.250,-82.045,-176.171,9.263,148.769
C07968=1158.379,373.003,-82.009,-176.172,9.259,148.769
C07969=1158.383,372.755,-81.973,-176.174,9.256,148.768
C07970=1158.387,372.508,-81.937,-176.176,9.251,148.768
C07971=1158.391,372.261,-81.902,-176.178,9.247,148.767
C07972=1158.395,372.013,-81.867,-176.180,9.243,148.767
C07973=1158.399,371.766,-81.831,-176.182,9.239,148.766
C07974=1158.403,371.518,-81.795,-176.184,9.236,148.766
C07975=1158.406,371.271,-81.759,-176.186,9.231,148.765
C07976=1158.411,371.024,-81.724,-176.188,9.228,148.765
C07977=1158.414,370.776,-81.689,-176.191,9.223,148.764
C07978=1158.418,370.529,-81.653,-176.193,9.220,148.764
C07979=1158.422,370.281,-81.617,-176.195,9.216,148.763
C07980=1158.426,370.033,-81.582,-176.197,9.212,148.763
C07981=1158.430,369.787,-81.546,-176.199,9.208,148.763
C07982=1158.434,369.539,-81.511,-176.201,9.204,148.762
C07983=1158.438,369.291,-81.476,-176.203,9.200,148.762
C07984=1158.442,369.044,-81.440,-176.206,9.196,148.761
C07985=1158.446,368.797,-81.405,-176.208,9.192,148.761
C07986=1158.450,368.549,-81.370,-176.210,9.188,148.760
C07987=1158.453,368.302,-81.334,-176.212,9.184,148.760
C07988=1158.457,368.054,-81.299,-176.215,9.180,148.760
C07989=1158.462,367.806,-81.264,-176.217,9.176,148.759
C07990=1158.466,367.559,-81.228,-176.219,9.172,148.759
C07991=1158.470,367.311,-81.192,-176.221,9.168,148.758
C07992=1158.474,367.065,-81.157,-176.224,9.164,148.758
C07993=1158.478,366.817,-81.122,-176.226,9.161,148.758
C07994=1158.481,366.569,-81.087,-176.228,9.156,148.757
C07995=1158.485,366.322,-81.051,-176.231,9.152,148.757
C07996=1158.490,366.074,-81.017,-176.233,9.149,148.756
C07997=1158.494,365.792,-80.977,-176.235,9.144,148.756
C07998=1158.498,365.508,-80.936,-176.238,9.140,148.756
C07999=1158.503,365.226,-80.896,-176.241,9.135,148.755
C08000=1158.508,364.943,-80.856,-176.244,9.130,148.755
C08001=1158.511,364.696,-80.821,-176.246,9.127,148.754
C08002=1158.515,364.448,-80.786,-176.249,9.123,148.754
C08003=1158.519,364.201,-80.751,-176.251,9.119,148.754
C08004=1158.523,363.953,-80.716,-176.253,9.115,148.753
C08005=1158.526,363.706,-80.681,-176.256,9.111,148.753
C08006=1158.531,363.459,-80.645,-176.258,9.107,148.753
C08007=1158.535,363.211,-80.611,-176.261,9.103,148.752
C08008=1158.538,362.963,-80.575,-176.263,9.100,148.752
C08009=1158.543,362.716,-80.541,-176.266,9.096,148.752
C08010=1158.546,362.468,-80.506,-176.269,9.091,148.751
C08011=1158.550,362.221,-80.471,-176.271,9.088,148.751
C08012=1158.554,361.973,-80.436,-176.273,9.084,148.751
C08013=1158.558,361.726,-80.401,-176.275,9.080,148.750
C08014=1158.563,361.478,-80.366,-176.278,9.076,148.750
C08015=1158.566,361.231,-80.331,-176.280,9.073,148.750
C08016=1158.570,360.984,-80.297,-176.283,9.068,148.749
C08017=1158.574,360.735,-80.262,-176.286,9.064,148.749
C08018=1158.578,360.488,-80.227,-176.288,9.061,148.749
C08019=1158.582,360.241,-80.192,-176.291,9.057,148.748
C08020=1158.586,359.993,-80.158,-176.293,9.053,148.748
C08021=1158.590,359.746,-80.123,-176.296,9.049,148.748
C08022=1158.594,359.498,-80.088,-176.298,9.046,148.747
C08023=1158.598,359.250,-80.053,-176.301,9.041,148.747
C08024=1158.602,359.003,-80.019,-176.303,9.038,148.747
C08025=1158.606,358.756,-79.984,-176.305,9.034,148.746
C08026=1158.610,358.508,-79.949,-176.308,9.030,148.746
C08027=1158.613,358.260,-79.915,-176.311,9.026,148.746
C08028=1158.618,358.012,-79.880,-176.312,9.023,148.746
C08029=1158.621,357.765,-79.845,-176.315,9.019,148.745
C08030=1158.625,357.518,-79.811,-176.318,9.015,148.745
C08031=1158.629,357.270,-79.776,-176.320,9.011,148.745
C08032=1158.634,357.022,-79.742,-176.322,9.008,148.744
C08033=1158.637,356.774,-79.707,-176.325,9.004,148.744
C08034=1158.641,356.527,-79.673,-176.328,9.000,148.744
C08035=1158.645,356.279,-79.638,-176.330,8.996,148.743
C08036=1158.649,356.032,-79.604,-176.332,8.993,148.743
C08037=1158.654,355.785,-79.569,-176.335,8.989,148.743
C08038=1158.657,355.537,-79.534,-176.337,8.985,148.743
C08039=1158.661,355.290,-79.500,-176.340,8.981,148.742
C08040=1158.665,355.042,-79.466,-176.342,8.978,148.742
C08041=1158.669,354.795,-79.432,-176.345,8.973,148.742
C08042=1158.673,354.546,-79.397,-176.347,8.970,148.741
C08043=1158.677,354.299,-79.363,-176.350,8.966,148.741
C08044=1158.681,354.051,-79.328,-176.352,8.962,148.741
C08045=1158.685,353.804,-79.294,-176.355,8.959,148.741
C08046=1158.689,353.557,-79.260,-176.357,8.955,148.740
C08047=1158.694,353.308,-79.226,-176.359,8.951,148.740
C08048=1158.697,353.061,-79.192,-176.362,8.947,148.740
C08049=1158.701,352.813,-79.157,-176.364,8.944,148.740
C08050=1158.705,352.566,-79.123,-176.367,8.940,148.739
C08051=1158.710,352.318,-79.089,-176.369,8.936,148.739
C08052=1158.713,352.070,-79.054,-176.372,8.932,148.739
C08053=1158.718,351.823,-79.020,-176.374,8.929,148.738
C08054=1158.721,351.575,-78.986,-176.377,8.926,148.738
C08055=1158.726,351.327,-78.952,-176.379,8.921,148.738
C08056=1158.729,351.080,-78.918,-176.381,8.918,148.738
C08057=1158.733,350.832,-78.884,-176.384,8.914,148.737
C08058=1158.737,350.585,-78.849,-176.387,8.911,148.737
C08059=1158.741,350.337,-78.816,-176.390,8.907,148.737
C08060=1158.745,350.089,-78.781,-176.391,8.903,148.736
C08061=1158.749,349.842,-78.748,-176.394,8.899,148.736
C08062=1158.754,349.594,-78.713,-176.397,8.896,148.736
C08063=1158.757,349.346,-78.680,-176.399,8.892,148.736
C08064=1158.761,349.099,-78.646,-176.402,8.888,148.735
C08065=1158.766,348.851,-78.611,-176.404,8.885,148.735
C08066=1158.769,348.603,-78.578,-176.407,8.880,148.735
C08067=1158.773,348.356,-78.544,-176.409,8.877,148.735
C08068=1158.778,348.108,-78.509,-176.411,8.874,148.734
C08069=1158.781,347.860,-78.476,-176.414,8.870,148.734
C08070=1158.785,347.613,-78.442,-176.416,8.866,148.734
C08071=1158.790,347.365,-78.408,-176.419,8.862,148.734
C08072=1158.794,347.118,-78.374,-176.422,8.859,148.733
C08073=1158.797,346.869,-78.341,-176.423,8.856,148.733
C08074=1158.802,346.622,-78.306,-176.426,8.851,148.733
C08075=1158.806,346.375,-78.272,-176.429,8.848,148.733
C08076=1158.810,346.127,-78.239,-176.432,8.844,148.732
C08077=1158.814,345.879,-78.205,-176.434,8.841,148.732
C08078=1158.818,345.631,-78.171,-176.436,8.837,148.732
C08079=1158.822,345.384,-78.138,-176.439,8.833,148.732
C08080=1158.826,345.136,-78.104,-176.441,8.830,148.731
C08081=1158.830,344.888,-78.070,-176.444,8.826,148.731
C08082=1158.834,344.641,-78.036,-176.447,8.823,148.731
C08083=1158.838,344.393,-78.003,-176.448,8.819,148.731
C08084=1158.842,344.146,-77.969,-176.451,8.815,148.730
C08085=1158.846,343.898,-77.936,-176.454,8.812,148.730
C08086=1158.850,343.649,-77.902,-176.456,8.808,148.730
C08087=1158.854,343.402,-77.868,-176.459,8.804,148.730
C08088=1158.858,343.154,-77.835,-176.461,8.801,148.729
C08089=1158.863,342.907,-77.802,-176.464,8.797,148.729
C08090=1158.866,342.660,-77.768,-176.466,8.794,148.729
C08091=1158.871,342.412,-77.734,-176.469,8.790,148.729
C08092=1158.875,342.163,-77.701,-176.471,8.786,148.728
C08093=1158.879,341.915,-77.668,-176.474,8.783,148.728
C08094=1158.883,341.668,-77.634,-176.476,8.780,148.728
C08095=1158.887,341.421,-77.601,-176.479,8.776,148.728
C08096=1158.891,341.173,-77.567,-176.481,8.772,148.728
C08097=1158.895,340.925,-77.534,-176.484,8.768,148.727
C08098=1158.899,340.678,-77.500,-176.486,8.765,148.727
C08099=1158.903,340.430,-77.467,-176.489,8.762,148.727
C08100=1158.907,340.181,-77.433,-176.492,8.758,148.727
C08101=1158.912,339.902,-77.396,-176.495,8.753,148.726
C08102=1158.917,339.622,-77.358,-176.497,8.750,148.726
C08103=1158.921,339.343,-77.320,-176.500,8.746,148.726
C08104=1158.926,339.063,-77.283,-176.503,8.742,148.726
C08105=1158.929,338.815,-77.249,-176.505,8.738,148.725
C08106=1158.933,338.567,-77.216,-176.508,8.735,148.725
C08107=1158.938,338.319,-77.183,-176.510,8.731,148.725
C08108=1158.942,338.072,-77.150,-176.513,8.727,148.725
C08109=1158.946,337.824,-77.117,-176.515,8.724,148.725
C08110=1158.950,337.576,-77.084,-176.518,8.721,148.724
C08111=1158.954,337.328,-77.050,-176.520,8.716,148.724
C08112=1158.958,337.081,-77.017,-176.523,8.713,148.724
C08113=1158.962,336.833,-76.984,-176.525,8.710,148.724
C08114=1158.967,336.585,-76.951,-176.528,8.706,148.724
C08115=1158.971,336.337,-76.918,-176.530,8.703,148.723
C08116=1158.975,336.090,-76.885,-176.533,8.699,148.723
C08117=1158.979,335.842,-76.852,-176.535,8.695,148.723
C08118=1158.982,335.595,-76.819,-176.538,8.692,148.723
C08119=1158.987,335.346,-76.787,-176.540,8.689,148.722
C08120=1158.991,335.098,-76.753,-176.543,8.684,148.722
C08121=1158.995,334.851,-76.720,-176.545,8.681,148.722
C08122=1158.999,334.603,-76.687,-176.548,8.678,148.722
C08123=1159.003,334.355,-76.654,-176.550,8.675,148.722
C08124=1159.008,334.108,-76.621,-176.553,8.671,148.721
C08125=1159.011,333.860,-76.588,-176.555,8.667,148.721
C08126=1159.015,333.612,-76.556,-176.558,8.664,148.721
C08127=1159.019,333.364,-76.523,-176.561,8.660,148.721
C08128=1159.024,333.116,-76.489,-176.563,8.657,148.721
C08129=1159.028,332.869,-76.456,-176.565,8.654,148.721
C08130=1159.031,332.621,-76.424,-176.568,8.649,148.720
C08131=1159.036,332.373,-76.391,-176.570,8.646,148.720
C08132=1159.040,332.125,-76.358,-176.573,8.643,148.720
C08133=1159.044,331.877,-76.325,-176.575,8.640,148.720
C08134=1159.048,331.629,-76.293,-176.578,8.636,148.719
C08135=1159.052,331.382,-76.260,-176.580,8.632,148.719
C08136=1159.056,331.134,-76.227,-176.583,8.629,148.719
C08137=1159.060,330.886,-76.194,-176.586,8.625,148.719
C08138=1159.064,330.638,-76.161,-176.588,8.622,148.719
C08139=1159.068,330.390,-76.129,-176.591,8.619,148.719
C08140=1159.072,330.142,-76.096,-176.593,8.614,148.718
C08141=1159.076,329.894,-76.063,-176.596,8.611,148.718
C08142=1159.081,329.647,-76.032,-176.598,8.608,148.718
C08143=1159.085,329.399,-75.998,-176.601,8.605,148.718
C08144=1159.089,329.151,-75.966,-176.604,8.601,148.718
C08145=1159.093,328.903,-75.933,-176.606,8.598,148.717
C08146=1159.097,328.655,-75.901,-176.608,8.594,148.717
C08147=1159.101,328.407,-75.868,-176.611,8.591,148.717
C08148=1159.105,328.159,-75.836,-176.613,8.587,148.717
C08149=1159.109,327.912,-75.803,-176.616,8.584,148.717
C08150=1159.114,327.664,-75.771,-176.618,8.581,148.717
C08151=1159.118,327.417,-75.738,-176.621,8.577,148.716
C08152=1159.122,327.168,-75.706,-176.624,8.573,148.716
C08153=1159.126,326.920,-75.674,-176.626,8.570,148.716
C08154=1159.130,326.672,-75.641,-176.628,8.567,148.716
C08155=1159.134,326.424,-75.609,-176.632,8.563,148.716
C08156=1159.138,326.177,-75.576,-176.634,8.560,148.716
C08157=1159.143,325.929,-75.544,-176.636,8.556,148.715
C08158=1159.146,325.681,-75.512,-176.639,8.553,148.715
C08159=1159.151,325.433,-75.479,-176.641,8.549,148.715
C08160=1159.154,325.185,-75.447,-176.644,8.546,148.715
C08161=1159.159,324.937,-75.414,-176.646,8.543,148.715
C08162=1159.163,324.690,-75.382,-176.649,8.539,148.715
C08163=1159.167,324.442,-75.350,-176.652,8.535,148.714
C08164=1159.171,324.194,-75.318,-176.654,8.532,148.714
C08165=1159.175,323.945,-75.285,-176.657,8.529,148.714
C08166=1159.179,323.698,-75.253,-176.659,8.526,148.714
C08167=1159.184,323.450,-75.221,-176.662,8.522,148.714
C08168=1159.188,323.202,-75.189,-176.664,8.518,148.714
C08169=1159.191,322.954,-75.157,-176.667,8.515,148.714
C08170=1159.196,322.706,-75.125,-176.669,8.512,148.713
C08171=1159.200,322.459,-75.093,-176.672,8.508,148.713
C08172=1159.204,322.211,-75.060,-176.674,8.505,148.713
C08173=1159.208,321.963,-75.028,-176.677,8.501,148.713
C08174=1159.212,321.714,-74.996,-176.680,8.499,148.713
C08175=1159.217,321.467,-74.964,-176.682,8.495,148.713
C08176=1159.220,321.219,-74.932,-176.685,8.491,148.712
C08177=1159.225,320.971,-74.900,-176.687,8.488,148.712
C08178=1159.228,320.723,-74.868,-176.690,8.485,148.712
C08179=1159.233,320.475,-74.837,-176.692,8.482,148.712
C08180=1159.237,320.227,-74.804,-176.695,8.477,148.712
C08181=1159.241,319.979,-74.772,-176.698,8.475,148.712
C08182=1159.245,319.732,-74.741,-176.700,8.471,148.712
C08183=1159.250,319.483,-74.709,-176.702,8.468,148.711
C08184=1159.253,319.235,-74.677,-176.705,8.465,148.711
C08185=1159.258,318.988,-74.645,-176.708,8.461,148.711
C08186=1159.262,318.740,-74.613,-176.710,8.458,148.711
C08187=1159.266,318.491,-74.581,-176.713,8.454,148.711
C08188=1159.270,318.244,-74.549,-176.715,8.451,148.711
C08189=1159.274,317.996,-74.518,-176.718,8.448,148.711
C08190=1159.278,317.748,-74.485,-176.720,8.444,148.710
C08191=1159.283,317.500,-74.454,-176.723,8.441,148.710
C08192=1159.286,317.252,-74.422,-176.726,8.438,148.710
C08193=1159.290,317.004,-74.390,-176.728,8.434,148.710
C08194=1159.295,316.756,-74.359,-176.731,8.430,148.710
C08195=1159.299,316.508,-74.327,-176.733,8.427,148.710
C08196=1159.303,316.261,-74.295,-176.736,8.424,148.710
C08197=1159.307,316.013,-74.263,-176.738,8.421,148.709
C08198=1159.311,315.765,-74.232,-176.741,8.418,148.709
C08199=1159.316,315.517,-74.200,-176.743,8.415,148.709
C08200=1159.320,315.268,-74.168,-176.746,8.410,148.709
C08201=1159.324,315.021,-74.137,-176.749,8.407,148.709
C08202=1159.328,314.773,-74.105,-176.751,8.404,148.709
C08203=1159.332,314.524,-74.074,-176.753,8.401,148.709
C08204=1159.336,314.277,-74.042,-176.756,8.398,148.709
C08205=1159.340,313.999,-74.007,-176.759,8.394,148.708
C08206=1159.345,313.723,-73.972,-176.762,8.390,148.708
C08207=1159.350,313.445,-73.936,-176.765,8.387,148.708
C08208=1159.355,313.168,-73.901,-176.768,8.383,148.708
C08209=1159.359,312.920,-73.870,-176.770,8.380,148.708
C08210=1159.363,312.672,-73.838,-176.773,8.376,148.708
C08211=1159.368,312.423,-73.806,-176.776,8.373,148.708
C08212=1159.372,312.176,-73.775,-176.778,8.369,148.708
C08213=1159.376,311.927,-73.744,-176.780,8.366,148.707
C08214=1159.380,311.680,-73.712,-176.783,8.363,148.707
C08215=1159.384,311.431,-73.681,-176.786,8.360,148.707
C08216=1159.389,311.184,-73.650,-176.788,8.356,148.707
C08217=1159.393,310.935,-73.619,-176.791,8.353,148.707
C08218=1159.397,310.688,-73.587,-176.793,8.349,148.707
C08219=1159.401,310.439,-73.556,-176.796,8.347,148.707
C08220=1159.405,310.192,-73.524,-176.799,8.343,148.707
C08221=1159.409,309.943,-73.493,-176.801,8.340,148.706
C08222=1159.414,309.696,-73.462,-176.804,8.336,148.706
C08223=1159.418,309.447,-73.431,-176.806,8.333,148.706
C08224=1159.422,309.200,-73.399,-176.809,8.330,148.706
C08225=1159.426,308.951,-73.368,-176.812,8.327,148.706
C08226=1159.431,308.703,-73.337,-176.814,8.324,148.706
C08227=1159.434,308.455,-73.306,-176.817,8.320,148.706
C08228=1159.439,308.207,-73.275,-176.819,8.317,148.706
C08229=1159.443,307.960,-73.243,-176.822,8.313,148.706
C08230=1159.446,307.712,-73.213,-176.825,8.310,148.706
C08231=1159.451,307.464,-73.182,-176.827,8.307,148.706
C08232=1159.455,307.216,-73.150,-176.830,8.304,148.705
C08233=1159.459,306.968,-73.119,-176.832,8.301,148.705
C08234=1159.464,306.720,-73.089,-176.835,8.298,148.705
C08235=1159.468,306.471,-73.057,-176.837,8.294,148.705
C08236=1159.472,306.224,-73.026,-176.840,8.290,148.705
C08237=1159.476,305.975,-72.995,-176.843,8.287,148.705
C08238=1159.480,305.727,-72.965,-176.845,8.284,148.705
C08239=1159.485,305.480,-72.934,-176.848,8.281,148.705
C08240=1159.489,305.231,-72.902,-176.850,8.278,148.705
C08241=1159.493,304.984,-72.871,-176.853,8.275,148.704
C08242=1159.498,304.736,-72.841,-176.855,8.272,148.705
C08243=1159.502,304.487,-72.809,-176.858,8.268,148.704
C08244=1159.506,304.239,-72.779,-176.861,8.265,148.704
C08245=1159.510,303.991,-72.748,-176.863,8.261,148.704
C08246=1159.514,303.743,-72.717,-176.866,8.258,148.704
C08247=1159.519,303.495,-72.686,-176.868,8.255,148.704
C08248=1159.523,303.247,-72.655,-176.871,8.252,148.704
C08249=1159.526,302.999,-72.625,-176.874,8.249,148.704
C08250=1159.531,302.751,-72.594,-176.876,8.246,148.704
C08251=1159.536,302.503,-72.563,-176.879,8.242,148.704
C08252=1159.540,302.254,-72.532,-176.882,8.239,148.704
C08253=1159.544,302.007,-72.502,-176.884,8.236,148.703
C08254=1159.548,301.759,-72.471,-176.887,8.233,148.704
C08255=1159.552,301.510,-72.440,-176.889,8.229,148.703
C08256=1159.556,301.262,-72.410,-176.892,8.226,148.703
C08257=1159.561,301.015,-72.379,-176.894,8.223,148.703
C08258=1159.565,300.767,-72.348,-176.897,8.220,148.703
C08259=1159.569,300.518,-72.318,-176.899,8.217,148.703
C08260=1159.573,300.270,-72.287,-176.903,8.213,148.703
C08261=1159.578,300.022,-72.257,-176.905,8.210,148.703
C08262=1159.581,299.773,-72.226,-176.908,8.207,148.703
C08263=1159.586,299.525,-72.196,-176.910,8.204,148.703
C08264=1159.591,299.277,-72.165,-176.913,8.201,148.703
C08265=1159.594,299.030,-72.135,-176.915,8.197,148.703
C08266=1159.598,298.781,-72.103,-176.918,8.194,148.703
C08267=1159.602,298.533,-72.073,-176.920,8.191,148.702
C08268=1159.607,298.285,-72.043,-176.923,8.188,148.702
C08269=1159.611,298.037,-72.013,-176.926,8.185,148.702
C08270=1159.616,297.789,-71.982,-176.928,8.182,148.702
C08271=1159.620,297.541,-71.951,-176.931,8.178,148.702
C08272=1159.624,297.293,-71.921,-176.934,8.175,148.702
C08273=1159.629,297.044,-71.891,-176.936,8.172,148.702
C08274=1159.632,296.797,-71.861,-176.939,8.169,148.702
C08275=1159.637,296.549,-71.830,-176.941,8.166,148.702
C08276=1159.640,296.300,-71.800,-176.944,8.163,148.702
C08277=1159.645,296.052,-71.769,-176.947,8.159,148.702
C08278=1159.649,295.804,-71.739,-176.949,8.156,148.702
C08279=1159.654,295.556,-71.709,-176.952,8.153,148.702
C08280=1159.658,295.308,-71.679,-176.954,8.150,148.702
C08281=1159.662,295.059,-71.648,-176.957,8.147,148.702
C08282=1159.666,294.811,-71.619,-176.959,8.144,148.702
C08283=1159.670,294.563,-71.588,-176.963,8.140,148.702
C08284=1159.675,294.315,-71.558,-176.965,8.137,148.701
C08285=1159.679,294.067,-71.528,-176.968,8.134,148.701
C08286=1159.683,293.819,-71.497,-176.970,8.131,148.701
C08287=1159.688,293.571,-71.468,-176.973,8.128,148.701
C08288=1159.692,293.322,-71.437,-176.976,8.125,148.701
C08289=1159.696,293.074,-71.407,-176.978,8.121,148.701
C08290=1159.700,292.826,-71.377,-176.981,8.118,148.701
C08291=1159.704,292.578,-71.346,-176.983,8.115,148.701
C08292=1159.708,292.330,-71.317,-176.986,8.112,148.701
C08293=1159.713,292.082,-71.287,-176.988,8.109,148.701
C08294=1159.717,291.834,-71.257,-176.991,8.106,148.701
C08295=1159.721,291.586,-71.227,-176.994,8.103,148.701
C08296=1159.725,291.338,-71.197,-176.996,8.100,148.701
C08297=1159.730,291.089,-71.167,-176.999,8.097,148.701
C08298=1159.733,290.841,-71.137,-177.001,8.094,148.701
C08299=1159.738,290.593,-71.107,-177.005,8.090,148.701
C08300=1159.743,290.344,-71.077,-177.007,8.087,148.701
C08301=1159.746,290.097,-71.047,-177.010,8.084,148.701
C08302=1159.751,289.848,-71.017,-177.012,8.080,148.700
C08303=1159.756,289.600,-70.987,-177.015,8.078,148.701
C08304=1159.759,289.352,-70.957,-177.018,8.075,148.701
C08305=1159.764,289.104,-70.928,-177.020,8.071,148.700
C08306=1159.768,288.856,-70.898,-177.023,8.068,148.700
C08307=1159.772,288.608,-70.867,-177.025,8.065,148.700
C08308=1159.777,288.359,-70.838,-177.028,8.062,148.700
C08309=1159.781,288.085,-70.805,-177.030,8.059,148.700
C08310=1159.786,287.809,-70.772,-177.034,8.055,148.700
C08311=1159.791,287.534,-70.739,-177.037,8.052,148.700
C08312=1159.796,287.259,-70.706,-177.039,8.048,148.700
C08313=1159.800,287.011,-70.677,-177.042,8.045,148.700
C08314=1159.804,286.763,-70.647,-177.045,8.042,148.700
C08315=1159.808,286.515,-70.617,-177.048,8.039,148.700
C08316=1159.812,286.267,-70.588,-177.050,8.036,148.700
C08317=1159.816,286.018,-70.558,-177.053,8.033,148.700
C08318=1159.821,285.770,-70.528,-177.055,8.030,148.700
C08319=1159.825,285.522,-70.499,-177.058,8.027,148.700
C08320=1159.830,285.273,-70.469,-177.061,8.024,148.700
C08321=1159.834,285.025,-70.440,-177.063,8.021,148.700
C08322=1159.838,284.777,-70.410,-177.066,8.018,148.700
C08323=1159.842,284.529,-70.380,-177.068,8.015,148.700
C08324=1159.846,284.281,-70.351,-177.071,8.012,148.700
C08325=1159.850,284.033,-70.321,-177.074,8.009,148.700
C08326=1159.855,283.785,-70.292,-177.076,8.006,148.700
C08327=1159.860,283.536,-70.262,-177.079,8.003,148.700
C08328=1159.864,283.288,-70.233,-177.082,8.000,148.700
C08329=1159.868,283.040,-70.203,-177.084,7.996,148.700
C08330=1159.873,282.792,-70.174,-177.087,7.993,148.700
C08331=1159.877,282.543,-70.145,-177.090,7.990,148.700
C08332=1159.881,282.294,-70.116,-177.092,7.988,148.700
C08333=1159.885,282.046,-70.086,-177.095,7.984,148.700
C08334=1159.890,281.798,-70.057,-177.097,7.981,148.700
C08335=1159.894,281.550,-70.028,-177.100,7.978,148.700
C08336=1159.899,281.302,-69.998,-177.103,7.975,148.700
C08337=1159.903,281.054,-69.969,-177.105,7.972,148.700
C08338=1159.907,280.806,-69.939,-177.108,7.969,148.700
C08339=1159.911,280.557,-69.910,-177.111,7.966,148.700
C08340=1159.916,280.308,-69.881,-177.113,7.963,148.700
C08341=1159.920,280.060,-69.852,-177.116,7.960,148.700
C08342=1159.924,279.813,-69.823,-177.119,7.957,148.700
C08343=1159.928,279.565,-69.794,-177.121,7.954,148.700
C08344=1159.932,279.316,-69.764,-177.124,7.951,148.700
C08345=1159.937,279.067,-69.735,-177.127,7.948,148.700
C08346=1159.941,278.819,-69.706,-177.129,7.945,148.700
C08347=1159.945,278.571,-69.677,-177.132,7.942,148.700
C08348=1159.950,278.323,-69.647,-177.135,7.939,148.700
C08349=1159.954,278.074,-69.619,-177.137,7.936,148.700
C08350=1159.958,277.826,-69.589,-177.140,7.933,148.700
C08351=1159.962,277.578,-69.560,-177.142,7.930,148.700
C08352=1159.966,277.329,-69.532,-177.145,7.927,148.700
C08353=1159.971,277.082,-69.503,-177.148,7.924,148.700
C08354=1159.975,276.833,-69.473,-177.151,7.921,148.700
C08355=1159.980,276.585,-69.444,-177.153,7.918,148.700
C08356=1159.984,276.336,-69.415,-177.156,7.915,148.700
C08357=1159.988,276.089,-69.386,-177.159,7.912,148.700
C08358=1159.993,275.840,-69.358,-177.161,7.909,148.700
C08359=1159.997,275.592,-69.328,-177.164,7.906,148.700
C08360=1160.001,275.343,-69.300,-177.167,7.903,148.700
C08361=1160.006,275.095,-69.270,-177.169,7.900,148.700
C08362=1160.010,274.847,-69.242,-177.172,7.897,148.700
C08363=1160.014,274.599,-69.213,-177.175,7.894,148.700
C08364=1160.018,274.350,-69.184,-177.177,7.892,148.700
C08365=1160.022,274.102,-69.156,-177.180,7.889,148.700
C08366=1160.027,273.854,-69.127,-177.182,7.886,148.700
C08367=1160.031,273.605,-69.097,-177.185,7.882,148.700
C08368=1160.036,273.357,-69.069,-177.187,7.879,148.700
C08369=1160.040,273.109,-69.040,-177.190,7.876,148.700
C08370=1160.044,272.860,-69.011,-177.193,7.873,148.700
C08371=1160.049,272.613,-68.982,-177.196,7.871,148.700
C08372=1160.053,272.364,-68.954,-177.198,7.868,148.700
C08373=1160.057,272.115,-68.925,-177.201,7.865,148.700
C08374=1160.061,271.867,-68.896,-177.204,7.861,148.700
C08375=1160.066,271.619,-68.868,-177.206,7.858,148.700
C08376=1160.070,271.371,-68.839,-177.209,7.855,148.700
C08377=1160.075,271.123,-68.810,-177.212,7.852,148.700
C08378=1160.079,270.874,-68.782,-177.215,7.850,148.700
C08379=1160.083,270.626,-68.753,-177.217,7.847,148.700
C08380=1160.087,270.378,-68.725,-177.220,7.844,148.700
C08381=1160.092,270.129,-68.696,-177.223,7.841,148.700
C08382=1160.096,269.880,-68.668,-177.225,7.838,148.700
C08383=1160.100,269.633,-68.639,-177.227,7.835,148.700
C08384=1160.105,269.384,-68.610,-177.230,7.832,148.700
C08385=1160.109,269.136,-68.583,-177.233,7.829,148.700
C08386=1160.114,268.887,-68.554,-177.236,7.826,148.700
C08387=1160.117,268.639,-68.525,-177.238,7.823,148.700
C08388=1160.122,268.391,-68.497,-177.241,7.820,148.701
C08389=1160.127,268.142,-68.468,-177.244,7.818,148.701
C08390=1160.131,267.894,-68.440,-177.247,7.815,148.701
C08391=1160.135,267.645,-68.411,-177.249,7.811,148.700
C08392=1160.139,267.397,-68.383,-177.252,7.808,148.701
C08393=1160.144,267.149,-68.355,-177.255,7.805,148.701
C08394=1160.148,266.901,-68.326,-177.257,7.802,148.701
C08395=1160.153,266.653,-68.298,-177.259,7.800,148.701
C08396=1160.157,266.404,-68.269,-177.262,7.797,148.701
C08397=1160.161,266.156,-68.242,-177.265,7.794,148.701
C08398=1160.165,265.907,-68.213,-177.268,7.791,148.701
C08399=1160.170,265.659,-68.185,-177.271,7.788,148.701
C08400=1160.174,265.410,-68.156,-177.273,7.786,148.701
C08401=1160.179,265.163,-68.129,-177.276,7.783,148.701
C08402=1160.183,264.914,-68.100,-177.279,7.780,148.701
C08403=1160.187,264.666,-68.072,-177.282,7.777,148.701
C08404=1160.192,264.417,-68.043,-177.284,7.774,148.701
C08405=1160.196,264.169,-68.016,-177.287,7.772,148.701
C08406=1160.200,263.920,-67.987,-177.289,7.768,148.701
C08407=1160.205,263.672,-67.959,-177.292,7.765,148.701
C08408=1160.209,263.424,-67.931,-177.294,7.762,148.701
C08409=1160.213,263.176,-67.903,-177.297,7.759,148.701
C08410=1160.218,262.926,-67.875,-177.300,7.757,148.701
C08411=1160.222,262.678,-67.847,-177.303,7.754,148.701
C08412=1160.226,262.430,-67.819,-177.305,7.751,148.701
C08413=1160.231,262.156,-67.788,-177.308,7.748,148.702
C08414=1160.236,261.884,-67.757,-177.311,7.745,148.702
C08415=1160.241,261.610,-67.726,-177.314,7.742,148.702
C08416=1160.246,261.338,-67.696,-177.318,7.738,148.702
C08417=1160.250,261.089,-67.667,-177.320,7.735,148.702
C08418=1160.255,260.840,-67.640,-177.323,7.732,148.702
C08419=1160.259,260.592,-67.612,-177.325,7.730,148.702
C08420=1160.263,260.344,-67.584,-177.328,7.727,148.702
C08421=1160.267,260.095,-67.556,-177.330,7.724,148.702
C08422=1160.272,259.846,-67.528,-177.333,7.721,148.702
C08423=1160.277,259.598,-67.500,-177.336,7.718,148.702
C08424=1160.280,259.350,-67.472,-177.339,7.715,148.702
C08425=1160.285,259.101,-67.445,-177.341,7.712,148.702
C08426=1160.289,258.853,-67.417,-177.344,7.710,148.702
C08427=1160.294,258.605,-67.389,-177.346,7.707,148.702
C08428=1160.298,258.356,-67.362,-177.350,7.705,148.703
C08429=1160.302,258.108,-67.333,-177.352,7.702,148.703
C08430=1160.307,257.860,-67.306,-177.355,7.699,148.703
C08431=1160.311,257.611,-67.279,-177.358,7.696,148.703
C08432=1160.315,257.363,-67.250,-177.361,7.693,148.703
C08433=1160.320,257.114,-67.222,-177.363,7.691,148.703
C08434=1160.325,256.866,-67.195,-177.366,7.688,148.703
C08435=1160.328,256.617,-67.167,-177.368,7.685,148.703
C08436=1160.333,256.369,-67.140,-177.371,7.682,148.703
C08437=1160.337,256.121,-67.112,-177.374,7.679,148.703
C08438=1160.341,255.872,-67.085,-177.377,7.676,148.703
C08439=1160.346,255.624,-67.057,-177.379,7.673,148.703
C08440=1160.350,255.375,-67.030,-177.382,7.671,148.703
C08441=1160.354,255.127,-67.002,-177.384,7.668,148.704
C08442=1160.360,254.878,-66.974,-177.387,7.665,148.704
C08443=1160.364,254.630,-66.946,-177.390,7.662,148.704
C08444=1160.368,254.381,-66.919,-177.393,7.659,148.704
C08445=1160.372,254.133,-66.891,-177.395,7.656,148.704
C08446=1160.377,253.885,-66.864,-177.398,7.654,148.704
C08447=1160.381,253.635,-66.836,-177.400,7.651,148.704
C08448=1160.385,253.388,-66.809,-177.403,7.648,148.704
C08449=1160.390,253.139,-66.782,-177.406,7.645,148.704
C08450=1160.394,252.891,-66.754,-177.409,7.643,148.704
C08451=1160.399,252.642,-66.726,-177.412,7.640,148.704
C08452=1160.403,252.393,-66.699,-177.414,7.637,148.705
C08453=1160.408,252.146,-66.672,-177.417,7.634,148.705
C08454=1160.412,251.897,-66.645,-177.420,7.632,148.705
C08455=1160.416,251.648,-66.617,-177.422,7.629,148.705
C08456=1160.421,251.399,-66.590,-177.425,7.626,148.705
C08457=1160.425,251.152,-66.562,-177.427,7.624,148.705
C08458=1160.429,250.903,-66.536,-177.430,7.621,148.705
C08459=1160.434,250.655,-66.509,-177.433,7.618,148.705
C08460=1160.438,250.406,-66.481,-177.436,7.615,148.705
C08461=1160.442,250.158,-66.454,-177.439,7.612,148.705
C08462=1160.447,249.909,-66.426,-177.441,7.610,148.705
C08463=1160.452,249.661,-66.399,-177.444,7.607,148.706
C08464=1160.456,249.412,-66.372,-177.447,7.604,148.706
C08465=1160.460,249.163,-66.345,-177.449,7.601,148.706
C08466=1160.465,248.915,-66.317,-177.452,7.598,148.706
C08467=1160.469,248.667,-66.291,-177.454,7.596,148.706
C08468=1160.473,248.419,-66.264,-177.457,7.593,148.706
C08469=1160.478,248.170,-66.237,-177.460,7.590,148.706
C08470=1160.482,247.921,-66.209,-177.463,7.588,148.706
C08471=1160.487,247.672,-66.182,-177.466,7.585,148.706
C08472=1160.491,247.424,-66.155,-177.468,7.582,148.706
C08473=1160.495,247.176,-66.129,-177.471,7.580,148.707
C08474=1160.500,246.927,-66.101,-177.474,7.577,148.707
C08475=1160.504,246.679,-66.074,-177.476,7.574,148.707
C08476=1160.509,246.430,-66.047,-177.479,7.571,148.707
C08477=1160.514,246.182,-66.020,-177.482,7.569,148.707
C08478=1160.517,245.933,-65.993,-177.485,7.566,148.707
C08479=1160.522,245.684,-65.966,-177.487,7.563,148.707
C08480=1160.526,245.436,-65.939,-177.490,7.560,148.707
C08481=1160.531,245.187,-65.912,-177.492,7.558,148.707
C08482=1160.535,244.939,-65.886,-177.495,7.555,148.707
C08483=1160.540,244.691,-65.859,-177.498,7.552,148.708
C08484=1160.544,244.442,-65.832,-177.501,7.549,148.708
C08485=1160.548,244.194,-65.805,-177.503,7.547,148.708
C08486=1160.553,243.945,-65.778,-177.506,7.544,148.708
C08487=1160.558,243.697,-65.751,-177.509,7.541,148.708
C08488=1160.561,243.449,-65.725,-177.512,7.538,148.708
C08489=1160.565,243.200,-65.697,-177.515,7.536,148.708
C08490=1160.570,242.950,-65.671,-177.517,7.534,148.708
C08491=1160.574,242.702,-65.644,-177.520,7.531,148.709
C08492=1160.579,242.454,-65.617,-177.523,7.528,148.709
C08493=1160.584,242.205,-65.590,-177.525,7.525,148.709
C08494=1160.588,241.957,-65.564,-177.527,7.523,148.709
C08495=1160.593,241.708,-65.537,-177.531,7.520,148.709
C08496=1160.597,241.459,-65.510,-177.533,7.517,148.709
C08497=1160.601,241.211,-65.484,-177.536,7.514,148.709
C08498=1160.606,240.963,-65.457,-177.538,7.512,148.709
C08499=1160.610,240.714,-65.431,-177.541,7.509,148.709
C08500=1160.615,240.466,-65.404,-177.544,7.507,148.710
C08501=1160.619,240.217,-65.377,-177.547,7.504,148.710
C08502=1160.623,239.969,-65.350,-177.549,7.502,148.710
C08503=1160.628,239.720,-65.324,-177.552,7.499,148.710
C08504=1160.632,239.472,-65.298,-177.555,7.496,148.710
C08505=1160.637,239.223,-65.271,-177.558,7.494,148.710
C08506=1160.641,238.974,-65.245,-177.560,7.491,148.710
C08507=1160.646,238.726,-65.218,-177.563,7.488,148.710
C08508=1160.650,238.477,-65.192,-177.566,7.485,148.711
C08509=1160.655,238.228,-65.165,-177.569,7.483,148.711
C08510=1160.658,237.980,-65.139,-177.571,7.480,148.711
C08511=1160.663,237.731,-65.112,-177.574,7.477,148.711
C08512=1160.668,237.484,-65.086,-177.576,7.475,148.711
C08513=1160.673,237.235,-65.060,-177.580,7.473,148.711
C08514=1160.677,236.986,-65.033,-177.582,7.470,148.712
C08515=1160.682,236.737,-65.007,-177.585,7.467,148.712
C08516=1160.686,236.489,-64.980,-177.587,7.465,148.712
C08517=1160.691,236.217,-64.952,-177.591,7.462,148.712
C08518=1160.696,235.946,-64.923,-177.593,7.459,148.712
C08519=1160.701,235.674,-64.894,-177.596,7.456,148.712
C08520=1160.705,235.402,-64.866,-177.600,7.453,148.712
C08521=1160.709,235.154,-64.839,-177.602,7.451,148.713
C08522=1160.714,234.905,-64.813,-177.605,7.448,148.713
C08523=1160.718,234.656,-64.787,-177.608,7.445,148.713
C08524=1160.722,234.408,-64.761,-177.610,7.443,148.713
C08525=1160.727,234.159,-64.734,-177.613,7.440,148.713
C08526=1160.731,233.910,-64.708,-177.616,7.437,148.713
C08527=1160.737,233.662,-64.682,-177.618,7.435,148.713
C08528=1160.741,233.413,-64.656,-177.621,7.432,148.714
C08529=1160.745,233.165,-64.630,-177.624,7.429,148.714
C08530=1160.750,232.916,-64.603,-177.627,7.428,148.714
C08531=1160.754,232.667,-64.578,-177.629,7.425,148.714
C08532=1160.758,232.419,-64.551,-177.632,7.422,148.714
C08533=1160.763,232.171,-64.526,-177.635,7.419,148.714
C08534=1160.768,231.922,-64.499,-177.638,7.417,148.715
C08535=1160.772,231.673,-64.474,-177.640,7.414,148.715
C08536=1160.776,231.425,-64.447,-177.643,7.411,148.715
C08537=1160.781,231.176,-64.421,-177.646,7.409,148.715
C08538=1160.786,230.928,-64.395,-177.649,7.406,148.715
C08539=1160.790,230.679,-64.370,-177.651,7.403,148.715
C08540=1160.794,230.430,-64.344,-177.654,7.402,148.716
C08541=1160.799,230.181,-64.317,-177.657,7.399,148.716
C08542=1160.803,229.933,-64.291,-177.660,7.396,148.716
C08543=1160.808,229.685,-64.266,-177.662,7.394,148.716
C08544=1160.812,229.436,-64.240,-177.665,7.391,148.716
C08545=1160.816,229.187,-64.214,-177.667,7.389,148.716
C08546=1160.821,228.938,-64.188,-177.671,7.386,148.717
C08547=1160.826,228.690,-64.162,-177.673,7.383,148.717
C08548=1160.830,228.441,-64.136,-177.675,7.381,148.717
C08549=1160.834,228.193,-64.110,-177.679,7.379,148.717
C08550=1160.839,227.944,-64.085,-177.682,7.376,148.717
C08551=1160.843,227.696,-64.059,-177.684,7.374,148.717
C08552=1160.848,227.447,-64.033,-177.687,7.371,148.717
C08553=1160.853,227.198,-64.007,-177.690,7.368,148.718
C08554=1160.857,226.949,-63.981,-177.692,7.366,148.718
C08555=1160.862,226.701,-63.956,-177.695,7.363,148.718
C08556=1160.866,226.452,-63.930,-177.698,7.360,148.718
C08557=1160.870,226.203,-63.904,-177.700,7.358,148.718
C08558=1160.875,225.955,-63.879,-177.703,7.356,148.718
C08559=1160.879,225.706,-63.853,-177.706,7.354,148.719
C08560=1160.883,225.458,-63.827,-177.708,7.351,148.719
C08561=1160.888,225.210,-63.802,-177.712,7.348,148.719
C08562=1160.892,224.961,-63.776,-177.714,7.346,148.719
C08563=1160.897,224.712,-63.751,-177.717,7.343,148.719
C08564=1160.901,224.462,-63.726,-177.720,7.340,148.719
C08565=1160.906,224.214,-63.700,-177.722,7.338,148.720
C08566=1160.910,223.966,-63.674,-177.725,7.336,148.720
C08567=1160.916,223.717,-63.648,-177.727,7.334,148.720
C08568=1160.920,223.468,-63.623,-177.730,7.331,148.720
C08569=1160.924,223.220,-63.597,-177.733,7.328,148.720
C08570=1160.929,222.971,-63.573,-177.736,7.326,148.721
C08571=1160.933,222.722,-63.547,-177.738,7.323,148.721
C08572=1160.937,222.474,-63.521,-177.741,7.321,148.721
C08573=1160.942,222.225,-63.496,-177.744,7.318,148.721
C08574=1160.946,221.977,-63.470,-177.747,7.316,148.721
C08575=1160.951,221.728,-63.446,-177.749,7.314,148.721
C08576=1160.955,221.479,-63.420,-177.752,7.311,148.722
C08577=1160.960,221.230,-63.394,-177.755,7.309,148.722
C08578=1160.965,220.982,-63.369,-177.758,7.306,148.722
C08579=1160.969,220.733,-63.344,-177.761,7.303,148.722
C08580=1160.974,220.485,-63.318,-177.763,7.301,148.722
C08581=1160.978,220.236,-63.293,-177.766,7.298,148.722
C08582=1160.983,219.986,-63.267,-177.768,7.296,148.723
C08583=1160.987,219.738,-63.242,-177.771,7.294,148.723
C08584=1160.991,219.490,-63.217,-177.774,7.291,148.723
C08585=1160.996,219.241,-63.192,-177.777,7.289,148.723
C08586=1161.000,218.992,-63.167,-177.779,7.286,148.723
C08587=1161.005,218.744,-63.142,-177.782,7.284,148.724
C08588=1161.010,218.495,-63.116,-177.785,7.281,148.724
C08589=1161.014,218.246,-63.090,-177.788,7.279,148.724
C08590=1161.018,217.998,-63.066,-177.790,7.276,148.724
C08591=1161.022,217.749,-63.041,-177.794,7.274,148.725
C08592=1161.028,217.500,-63.016,-177.796,7.272,148.725
C08593=1161.032,217.251,-62.990,-177.799,7.269,148.725
C08594=1161.037,217.003,-62.965,-177.801,7.267,148.725
C08595=1161.040,216.754,-62.940,-177.804,7.264,148.725
C08596=1161.046,216.505,-62.916,-177.807,7.262,148.726
C08597=1161.050,216.256,-62.890,-177.809,7.259,148.726
C08598=1161.055,216.008,-62.865,-177.812,7.258,148.726
C08599=1161.058,215.759,-62.840,-177.815,7.255,148.726
C08600=1161.064,215.511,-62.815,-177.818,7.252,148.726
C08601=1161.068,215.262,-62.790,-177.820,7.250,148.727
C08602=1161.073,215.013,-62.765,-177.823,7.247,148.727
C08603=1161.077,214.764,-62.741,-177.826,7.245,148.727
C08604=1161.082,214.516,-62.715,-177.829,7.242,148.727
C08605=1161.086,214.266,-62.690,-177.831,7.241,148.727
C08606=1161.090,214.019,-62.665,-177.834,7.238,148.727
C08607=1161.095,213.770,-62.641,-177.837,7.236,148.728
C08608=1161.100,213.520,-62.616,-177.839,7.233,148.728
C08609=1161.104,213.273,-62.591,-177.842,7.231,148.728
C08610=1161.108,213.023,-62.566,-177.845,7.228,148.728
C08611=1161.114,212.774,-62.541,-177.848,7.226,148.729
C08612=1161.117,212.525,-62.517,-177.850,7.223,148.729
C08613=1161.122,212.277,-62.491,-177.853,7.222,148.729
C08614=1161.127,212.029,-62.467,-177.856,7.219,148.729
C08615=1161.131,211.779,-62.442,-177.859,7.216,148.730
C08616=1161.136,211.531,-62.417,-177.861,7.214,148.730
C08617=1161.140,211.282,-62.392,-177.865,7.211,148.730
C08618=1161.145,211.034,-62.368,-177.867,7.209,148.730
C08619=1161.150,210.785,-62.343,-177.870,7.207,148.730
C08620=1161.154,210.536,-62.319,-177.872,7.205,148.731
C08621=1161.159,210.265,-62.292,-177.875,7.202,148.731
C08622=1161.164,209.995,-62.265,-177.878,7.199,148.731
C08623=1161.169,209.724,-62.238,-177.881,7.197,148.731
C08624=1161.174,209.454,-62.211,-177.884,7.195,148.732
C08625=1161.178,209.205,-62.186,-177.887,7.192,148.732
C08626=1161.183,208.956,-62.162,-177.890,7.190,148.732
C08627=1161.188,208.708,-62.138,-177.892,7.187,148.732
C08628=1161.192,208.459,-62.113,-177.895,7.185,148.732
C08629=1161.196,208.211,-62.088,-177.898,7.182,148.733
C08630=1161.201,207.962,-62.064,-177.900,7.181,148.733
C08631=1161.205,207.713,-62.039,-177.903,7.178,148.733
C08632=1161.210,207.464,-62.015,-177.906,7.176,148.733
C08633=1161.215,207.216,-61.990,-177.909,7.173,148.733
C08634=1161.219,206.966,-61.965,-177.911,7.171,148.734
C08635=1161.224,206.718,-61.941,-177.914,7.168,148.734
C08636=1161.228,206.469,-61.917,-177.917,7.167,148.734
C08637=1161.232,206.220,-61.892,-177.920,7.164,148.734
C08638=1161.237,205.971,-61.868,-177.922,7.162,148.735
C08639=1161.242,205.723,-61.844,-177.925,7.159,148.735
C08640=1161.247,205.474,-61.819,-177.928,7.157,148.735
C08641=1161.251,205.225,-61.795,-177.931,7.154,148.735
C08642=1161.256,204.976,-61.770,-177.933,7.152,148.736
C08643=1161.260,204.727,-61.746,-177.935,7.150,148.736
C08644=1161.265,204.479,-61.722,-177.939,7.148,148.736
C08645=1161.269,204.230,-61.697,-177.941,7.146,148.736
C08646=1161.274,203.981,-61.673,-177.944,7.143,148.736
C08647=1161.278,203.733,-61.649,-177.947,7.141,148.737
C08648=1161.283,203.484,-61.624,-177.950,7.138,148.737
C08649=1161.287,203.234,-61.601,-177.952,7.137,148.737
C08650=1161.292,202.986,-61.577,-177.955,7.134,148.737
C08651=1161.297,202.737,-61.552,-177.958,7.132,148.738
C08652=1161.301,202.489,-61.528,-177.961,7.129,148.738
C08653=1161.306,202.240,-61.504,-177.963,7.127,148.738
C08654=1161.310,201.990,-61.480,-177.966,7.125,148.739
C08655=1161.315,201.742,-61.455,-177.969,7.122,148.739
C08656=1161.319,201.493,-61.431,-177.971,7.121,148.739
C08657=1161.324,201.245,-61.407,-177.974,7.118,148.739
C08658=1161.329,200.996,-61.383,-177.977,7.116,148.739
C08659=1161.333,200.747,-61.359,-177.980,7.113,148.740
C08660=1161.337,200.498,-61.335,-177.982,7.111,148.740
C08661=1161.342,200.250,-61.311,-177.985,7.109,148.740
C08662=1161.347,200.000,-61.287,-177.988,7.107,148.740
C08663=1161.351,199.752,-61.263,-177.990,7.105,148.741
C08664=1161.356,199.504,-61.239,-177.993,7.102,148.741
C08665=1161.360,199.254,-61.215,-177.996,7.100,148.741
C08666=1161.364,199.005,-61.191,-177.999,7.098,148.741
C08667=1161.370,198.756,-61.167,-178.001,7.095,148.742
C08668=1161.374,198.508,-61.143,-178.005,7.093,148.742
C08669=1161.379,198.259,-61.119,-178.007,7.091,148.742
C08670=1161.383,198.010,-61.095,-178.009,7.089,148.742
C08671=1161.388,197.762,-61.071,-178.013,7.086,148.743
C08672=1161.392,197.512,-61.048,-178.015,7.084,148.743
C08673=1161.397,197.263,-61.023,-178.018,7.082,148.743
C08674=1161.402,197.014,-61.000,-178.020,7.080,148.743
C08675=1161.406,196.766,-60.975,-178.023,7.078,148.744
C08676=1161.411,196.517,-60.952,-178.026,7.075,148.744
C08677=1161.415,196.269,-60.928,-178.029,7.073,148.744
C08678=1161.420,196.019,-60.905,-178.032,7.071,148.744
C08679=1161.424,195.771,-60.881,-178.034,7.069,148.745
C08680=1161.429,195.522,-60.857,-178.037,7.067,148.745
C08681=1161.433,195.274,-60.833,-178.040,7.064,148.745
C08682=1161.438,195.025,-60.810,-178.042,7.062,148.745
C08683=1161.442,194.776,-60.786,-178.045,7.059,148.746
C08684=1161.448,194.527,-60.762,-178.048,7.058,148.746
C08685=1161.452,194.277,-60.738,-178.050,7.056,148.746
C08686=1161.456,194.029,-60.714,-178.054,7.053,148.747
C08687=1161.461,193.780,-60.691,-178.056,7.051,148.747
C08688=1161.466,193.531,-60.667,-178.059,7.048,148.747
C08689=1161.470,193.282,-60.643,-178.062,7.047,148.747
C08690=1161.475,193.033,-60.620,-178.064,7.045,148.748
C08691=1161.479,192.784,-60.596,-178.067,7.042,148.748
C08692=1161.484,192.536,-60.572,-178.070,7.040,148.748
C08693=1161.489,192.287,-60.549,-178.072,7.038,148.749
C08694=1161.493,192.038,-60.526,-178.075,7.035,148.749
C08695=1161.498,191.789,-60.502,-178.078,7.034,148.749
C08696=1161.502,191.540,-60.478,-178.081,7.031,148.749
C08697=1161.507,191.291,-60.455,-178.083,7.029,148.749
C08698=1161.511,191.042,-60.432,-178.086,7.027,148.750
C08699=1161.515,190.794,-60.408,-178.089,7.024,148.750
C08700=1161.520,190.545,-60.385,-178.092,7.022,148.750
C08701=1161.525,190.296,-60.361,-178.094,7.021,148.751
C08702=1161.530,190.047,-60.338,-178.097,7.018,148.751
C08703=1161.535,189.799,-60.315,-178.100,7.016,148.751
C08704=1161.539,189.550,-60.291,-178.102,7.014,148.751
C08705=1161.544,189.301,-60.268,-178.105,7.011,148.752
C08706=1161.549,189.052,-60.244,-178.108,7.010,148.752
C08707=1161.553,188.803,-60.221,-178.111,7.008,148.752
C08708=1161.558,188.554,-60.197,-178.114,7.005,148.753
C08709=1161.562,188.305,-60.175,-178.116,7.003,148.753
C08710=1161.567,188.056,-60.151,-178.119,7.001,148.753
C08711=1161.571,187.807,-60.128,-178.122,6.999,148.753
C08712=1161.576,187.558,-60.105,-178.124,6.997,148.754
C08713=1161.580,187.310,-60.081,-178.127,6.994,148.754
C08714=1161.585,187.061,-60.057,-178.130,6.992,148.754
C08715=1161.589,186.812,-60.034,-178.132,6.990,148.754
C08716=1161.594,186.564,-60.011,-178.136,6.988,148.755
C08717=1161.599,186.315,-59.988,-178.138,6.986,148.755
C08718=1161.604,186.066,-59.965,-178.141,6.984,148.755
C08719=1161.608,185.817,-59.942,-178.144,6.981,148.756
C08720=1161.613,185.568,-59.919,-178.146,6.980,148.756
C08721=1161.617,185.319,-59.895,-178.149,6.978,148.756
C08722=1161.622,185.070,-59.872,-178.152,6.975,148.756
C08723=1161.626,184.821,-59.850,-178.155,6.973,148.757
C08724=1161.631,184.572,-59.827,-178.157,6.971,148.757
C08725=1161.636,184.303,-59.801,-178.161,6.969,148.757
C08726=1161.642,184.033,-59.776,-178.163,6.967,148.758
C08727=1161.646,183.763,-59.751,-178.166,6.964,148.758
C08728=1161.651,183.493,-59.726,-178.169,6.962,148.758
C08729=1161.656,183.245,-59.703,-178.172,6.960,148.759
C08730=1161.660,182.996,-59.680,-178.175,6.958,148.759
C08731=1161.665,182.747,-59.657,-178.177,6.956,148.759
C08732=1161.670,182.498,-59.634,-178.180,6.953,148.759
C08733=1161.674,182.249,-59.612,-178.183,6.952,148.760
C08734=1161.679,182.001,-59.589,-178.185,6.950,148.760
C08735=1161.684,181.752,-59.565,-178.188,6.947,148.760
C08736=1161.688,181.503,-59.543,-178.191,6.945,148.761
C08737=1161.693,181.253,-59.520,-178.194,6.943,148.761
C08738=1161.697,181.004,-59.497,-178.196,6.942,148.761
C08739=1161.702,180.756,-59.474,-178.199,6.939,148.761
C08740=1161.707,180.507,-59.451,-178.202,6.937,148.762
C08741=1161.711,180.258,-59.429,-178.204,6.935,148.762
C08742=1161.716,180.009,-59.405,-178.208,6.933,148.763
C08743=1161.720,179.760,-59.383,-178.210,6.930,148.763
C08744=1161.726,179.511,-59.360,-178.213,6.929,148.763
C08745=1161.729,179.262,-59.338,-178.215,6.927,148.763
C08746=1161.734,179.013,-59.314,-178.219,6.924,148.764
C08747=1161.740,178.764,-59.292,-178.221,6.922,148.764
C08748=1161.744,178.516,-59.269,-178.224,6.921,148.764
C08749=1161.748,178.267,-59.246,-178.227,6.918,148.765
C08750=1161.753,178.017,-59.224,-178.229,6.916,148.765
C08751=1161.758,177.769,-59.201,-178.232,6.914,148.765
C08752=1161.762,177.520,-59.178,-178.234,6.912,148.765
C08753=1161.767,177.271,-59.155,-178.238,6.910,148.766
C08754=1161.771,177.022,-59.133,-178.240,6.908,148.766
C08755=1161.777,176.773,-59.110,-178.243,6.906,148.767
C08756=1161.780,176.524,-59.088,-178.245,6.904,148.767
C08757=1161.786,176.275,-59.065,-178.248,6.902,148.767
C08758=1161.790,176.026,-59.043,-178.251,6.900,148.767
C08759=1161.794,175.777,-59.021,-178.254,6.898,148.768
C08760=1161.799,175.528,-58.997,-178.257,6.896,148.768
C08761=1161.804,175.279,-58.975,-178.259,6.893,148.768
C08762=1161.809,175.030,-58.952,-178.262,6.892,148.769
C08763=1161.813,174.781,-58.930,-178.265,6.890,148.769
C08764=1161.818,174.533,-58.907,-178.267,6.888,148.769
C08765=1161.822,174.283,-58.885,-178.271,6.886,148.770
C08766=1161.826,174.035,-58.862,-178.273,6.884,148.770
C08767=1161.832,173.786,-58.840,-178.276,6.882,148.770
C08768=1161.836,173.536,-58.818,-178.278,6.880,148.771
C08769=1161.842,173.288,-58.795,-178.282,6.877,148.771
C08770=1161.846,173.039,-58.773,-178.284,6.876,148.771
C08771=1161.850,172.790,-58.750,-178.286,6.874,148.771
C08772=1161.855,172.541,-58.728,-178.289,6.872,148.772
C08773=1161.860,172.292,-58.706,-178.292,6.869,148.772
C08774=1161.864,172.044,-58.683,-178.295,6.868,148.773
C08775=1161.869,171.794,-58.661,-178.298,6.866,148.773
C08776=1161.874,171.545,-58.639,-178.300,6.864,148.773
C08777=1161.878,171.297,-58.616,-178.303,6.862,148.773
C08778=1161.883,171.047,-58.594,-178.306,6.859,148.774
C08779=1161.888,170.798,-58.572,-178.309,6.858,148.774
C08780=1161.892,170.549,-58.550,-178.311,6.856,148.774
C08781=1161.896,170.300,-58.527,-178.314,6.854,148.775
C08782=1161.902,170.051,-58.505,-178.316,6.852,148.775
C08783=1161.906,169.802,-58.483,-178.320,6.849,148.775
C08784=1161.911,169.553,-58.461,-178.322,6.848,148.776
C08785=1161.916,169.304,-58.438,-178.325,6.846,148.776
C08786=1161.921,169.056,-58.416,-178.328,6.844,148.776
C08787=1161.925,168.806,-58.394,-178.330,6.842,148.777
C08788=1161.930,168.558,-58.372,-178.333,6.840,148.777
C08789=1161.934,168.308,-58.350,-178.336,6.838,148.777
C08790=1161.940,168.059,-58.328,-178.338,6.836,148.778
C08791=1161.943,167.811,-58.305,-178.341,6.834,148.778
C08792=1161.948,167.562,-58.284,-178.344,6.833,148.778
C08793=1161.953,167.313,-58.262,-178.347,6.830,148.779
C08794=1161.958,167.064,-58.239,-178.350,6.828,148.779
C08795=1161.962,166.814,-58.217,-178.352,6.826,148.779
C08796=1161.967,166.566,-58.196,-178.355,6.824,148.780
C08797=1161.972,166.316,-58.174,-178.357,6.823,148.780
C08798=1161.976,166.068,-58.152,-178.361,6.820,148.780
C08799=1161.981,165.819,-58.130,-178.363,6.818,148.781
C08800=1161.986,165.570,-58.108,-178.366,6.817,148.781
C08801=1161.991,165.320,-58.085,-178.369,6.815,148.781
C08802=1161.996,165.072,-58.064,-178.371,6.813,148.782
C08803=1162.000,164.822,-58.042,-178.374,6.811,148.782
C08804=1162.005,164.574,-58.020,-178.377,6.808,148.782
C08805=1162.009,164.324,-57.998,-178.380,6.807,148.783
C08806=1162.014,164.076,-57.976,-178.382,6.805,148.783
C08807=1162.019,163.827,-57.955,-178.385,6.803,148.783
C08808=1162.023,163.578,-57.933,-178.388,6.801,148.784
C08809=1162.028,163.329,-57.911,-178.390,6.800,148.784
C08810=1162.032,163.080,-57.889,-178.394,6.797,148.785
C08811=1162.037,162.831,-57.867,-178.396,6.795,148.785
C08812=1162.041,162.582,-57.845,-178.399,6.793,148.785
C08813=1162.046,162.333,-57.823,-178.401,6.792,148.785
C08814=1162.051,162.084,-57.802,-178.404,6.790,148.786
C08815=1162.056,161.834,-57.780,-178.407,6.788,148.786
C08816=1162.060,161.586,-57.759,-178.410,6.785,148.787
C08817=1162.065,161.336,-57.737,-178.413,6.784,148.787
C08818=1162.070,161.088,-57.715,-178.415,6.782,148.787
C08819=1162.074,160.839,-57.693,-178.418,6.780,148.788
C08820=1162.079,160.590,-57.671,-178.421,6.779,148.788
C08821=1162.084,160.341,-57.650,-178.423,6.776,148.788
C08822=1162.089,160.092,-57.629,-178.426,6.775,148.789
C08823=1162.093,159.843,-57.607,-178.428,6.773,148.789
C08824=1162.098,159.594,-57.585,-178.432,6.770,148.789
C08825=1162.102,159.344,-57.564,-178.434,6.769,148.790
C08826=1162.107,159.095,-57.542,-178.437,6.767,148.790
C08827=1162.112,158.847,-57.520,-178.440,6.765,148.790
C08828=1162.116,158.597,-57.498,-178.442,6.763,148.791
C08829=1162.121,158.328,-57.475,-178.446,6.761,148.791
C08830=1162.127,158.060,-57.452,-178.448,6.759,148.792
C08831=1162.132,157.791,-57.429,-178.451,6.757,148.792
C08832=1162.137,157.522,-57.406,-178.454,6.755,148.792
C08833=1162.142,157.272,-57.384,-178.457,6.753,148.793
C08834=1162.147,157.023,-57.363,-178.460,6.751,148.793
C08835=1162.151,156.775,-57.341,-178.462,6.750,148.793
C08836=1162.156,156.526,-57.320,-178.465,6.748,148.794
C08837=1162.160,156.276,-57.298,-178.468,6.746,148.794
C08838=1162.165,156.028,-57.277,-178.471,6.744,148.795
C08839=1162.170,155.778,-57.256,-178.473,6.743,148.795
C08840=1162.174,155.529,-57.234,-178.477,6.740,148.795
C08841=1162.180,155.280,-57.213,-178.479,6.738,148.796
C08842=1162.184,155.032,-57.192,-178.482,6.737,148.796
C08843=1162.189,154.782,-57.171,-178.484,6.734,148.796
C08844=1162.193,154.533,-57.149,-178.487,6.733,148.797
C08845=1162.198,154.284,-57.128,-178.490,6.731,148.797
C08846=1162.203,154.035,-57.107,-178.492,6.729,148.797
C08847=1162.208,153.786,-57.086,-178.495,6.728,148.798
C08848=1162.212,153.537,-57.064,-178.498,6.726,148.798
C08849=1162.217,153.287,-57.043,-178.500,6.724,148.798
C08850=1162.222,153.039,-57.021,-178.503,6.722,148.799
C08851=1162.226,152.790,-57.001,-178.506,6.720,148.799
C08852=1162.231,152.541,-56.979,-178.509,6.718,148.800
C08853=1162.236,152.291,-56.958,-178.512,6.716,148.800
C08854=1162.240,152.043,-56.936,-178.514,6.715,148.800
C08855=1162.245,151.794,-56.916,-178.517,6.713,148.801
C08856=1162.250,151.544,-56.895,-178.520,6.711,148.801
C08857=1162.255,151.296,-56.873,-178.522,6.709,148.802
C08858=1162.259,151.046,-56.852,-178.525,6.708,148.802
C08859=1162.264,150.797,-56.831,-178.528,6.706,148.802
C08860=1162.269,150.548,-56.809,-178.531,6.704,148.803
C08861=1162.274,150.299,-56.789,-178.533,6.702,148.803
C08862=1162.279,150.050,-56.768,-178.536,6.701,148.803
C08863=1162.284,149.801,-56.746,-178.539,6.699,148.804
C08864=1162.287,149.552,-56.726,-178.541,6.697,148.804
C08865=1162.293,149.302,-56.705,-178.544,6.695,148.805
C08866=1162.298,149.054,-56.683,-178.547,6.693,148.805
C08867=1162.302,148.805,-56.663,-178.550,6.691,148.805
C08868=1162.307,148.556,-56.642,-178.553,6.689,148.806
C08869=1162.312,148.307,-56.621,-178.555,6.688,148.806
C08870=1162.316,148.058,-56.600,-178.558,6.686,148.806
C08871=1162.321,147.808,-56.578,-178.561,6.684,148.807
C08872=1162.325,147.559,-56.558,-178.564,6.682,148.807
C08873=1162.331,147.310,-56.537,-178.566,6.681,148.808
C08874=1162.335,147.062,-56.516,-178.569,6.679,148.808
C08875=1162.340,146.812,-56.495,-178.572,6.677,148.808
C08876=1162.344,146.563,-56.475,-178.574,6.676,148.809
C08877=1162.350,146.314,-56.454,-178.577,6.674,148.809
C08878=1162.354,146.065,-56.433,-178.580,6.672,148.810
C08879=1162.359,145.816,-56.412,-178.582,6.670,148.810
C08880=1162.364,145.567,-56.392,-178.585,6.669,148.810
C08881=1162.368,145.318,-56.370,-178.588,6.667,148.811
C08882=1162.373,145.068,-56.349,-178.591,6.665,148.811
C08883=1162.377,144.819,-56.329,-178.593,6.663,148.811
C08884=1162.382,144.570,-56.308,-178.596,6.662,148.812
C08885=1162.387,144.321,-56.287,-178.599,6.660,148.812
C08886=1162.392,144.072,-56.267,-178.601,6.658,148.813
C08887=1162.397,143.823,-56.246,-178.604,6.656,148.813
C08888=1162.401,143.574,-56.225,-178.607,6.655,148.813
C08889=1162.406,143.325,-56.205,-178.609,6.653,148.814
C08890=1162.411,143.076,-56.184,-178.612,6.651,148.814
C08891=1162.416,142.827,-56.163,-178.615,6.649,148.815
C08892=1162.420,142.578,-56.143,-178.618,6.648,148.815
C08893=1162.425,142.329,-56.122,-178.620,6.646,148.815
C08894=1162.430,142.079,-56.101,-178.623,6.644,148.816
C08895=1162.434,141.830,-56.081,-178.626,6.643,148.816
C08896=1162.440,141.581,-56.060,-178.628,6.641,148.816
C08897=1162.444,141.332,-56.040,-178.631,6.639,148.817
C08898=1162.448,141.083,-56.019,-178.634,6.637,148.817
C08899=1162.454,140.834,-55.998,-178.637,6.636,148.818
C08900=1162.458,140.585,-55.978,-178.639,6.634,148.818
C08901=1162.463,140.336,-55.957,-178.642,6.632,148.818
C08902=1162.468,140.086,-55.937,-178.645,6.631,148.819
C08903=1162.472,139.837,-55.917,-178.648,6.629,148.819
C08904=1162.478,139.588,-55.896,-178.651,6.627,148.820
C08905=1162.482,139.339,-55.876,-178.653,6.626,148.820
C08906=1162.486,139.090,-55.855,-178.656,6.624,148.821
C08907=1162.492,138.841,-55.834,-178.659,6.622,148.821
C08908=1162.496,138.592,-55.814,-178.661,6.620,148.821
C08909=1162.501,138.342,-55.794,-178.664,6.619,148.822
C08910=1162.505,138.093,-55.774,-178.667,6.617,148.822
C08911=1162.510,137.844,-55.753,-178.669,6.615,148.822
C08912=1162.515,137.595,-55.733,-178.672,6.614,148.823
C08913=1162.520,137.346,-55.713,-178.675,6.612,148.823
C08914=1162.525,137.097,-55.692,-178.678,6.610,148.824
C08915=1162.530,136.848,-55.672,-178.680,6.608,148.824
C08916=1162.534,136.599,-55.652,-178.683,6.607,148.824
C08917=1162.539,136.350,-55.632,-178.686,6.605,148.825
C08918=1162.543,136.101,-55.612,-178.689,6.603,148.825
C08919=1162.549,135.851,-55.591,-178.692,6.602,148.826
C08920=1162.553,135.602,-55.571,-178.694,6.600,148.826
C08921=1162.558,135.353,-55.551,-178.697,6.598,148.827
C08922=1162.562,135.104,-55.530,-178.700,6.597,148.827
C08923=1162.568,134.854,-55.510,-178.702,6.595,148.827
C08924=1162.573,134.606,-55.490,-178.705,6.593,148.828
C08925=1162.577,134.357,-55.470,-178.708,6.591,148.828
C08926=1162.582,134.107,-55.450,-178.711,6.590,148.829
C08927=1162.586,133.858,-55.430,-178.713,6.588,148.829
C08928=1162.591,133.609,-55.409,-178.715,6.587,148.829
C08929=1162.596,133.359,-55.389,-178.718,6.585,148.830
C08930=1162.601,133.111,-55.369,-178.721,6.584,148.830
C08931=1162.606,132.862,-55.349,-178.724,6.582,148.831
C08932=1162.610,132.613,-55.329,-178.727,6.580,148.831
C08933=1162.615,132.344,-55.308,-178.729,6.579,148.832
C08934=1162.621,132.075,-55.286,-178.733,6.576,148.832
C08935=1162.626,131.807,-55.264,-178.736,6.575,148.833
C08936=1162.631,131.538,-55.243,-178.739,6.573,148.833
C08937=1162.636,131.289,-55.222,-178.741,6.571,148.833
C08938=1162.641,131.040,-55.203,-178.744,6.570,148.834
C08939=1162.646,130.791,-55.183,-178.747,6.568,148.834
C08940=1162.650,130.542,-55.163,-178.749,6.566,148.835
C08941=1162.655,130.292,-55.143,-178.752,6.564,148.835
C08942=1162.659,130.043,-55.123,-178.755,6.564,148.836
C08943=1162.664,129.794,-55.103,-178.757,6.562,148.836
C08944=1162.669,129.545,-55.083,-178.760,6.560,148.836
C08945=1162.674,129.296,-55.064,-178.763,6.559,148.837
C08946=1162.678,129.047,-55.043,-178.766,6.557,148.837
C08947=1162.683,128.797,-55.024,-178.768,6.555,148.837
C08948=1162.689,128.549,-55.004,-178.771,6.554,148.838
C08949=1162.693,128.300,-54.984,-178.774,6.552,148.838
C08950=1162.698,128.050,-54.964,-178.776,6.550,148.839
C08951=1162.702,127.800,-54.945,-178.780,6.549,148.839
C08952=1162.707,127.552,-54.925,-178.782,6.547,148.840
C08953=1162.712,127.303,-54.905,-178.784,6.546,148.840
C08954=1162.717,127.053,-54.885,-178.787,6.544,148.841
C08955=1162.721,126.804,-54.865,-178.790,6.543,148.841
C08956=1162.727,126.555,-54.846,-178.793,6.541,148.841
C08957=1162.731,126.306,-54.826,-178.795,6.539,148.842
C08958=1162.736,126.057,-54.806,-178.798,6.538,148.842
C08959=1162.741,125.808,-54.786,-178.801,6.536,148.843
C08960=1162.746,125.558,-54.767,-178.804,6.534,148.843
C08961=1162.751,125.309,-54.747,-178.807,6.533,148.843
C08962=1162.756,125.059,-54.727,-178.809,6.532,148.844
C08963=1162.761,124.811,-54.707,-178.811,6.530,148.844
C08964=1162.765,124.561,-54.688,-178.814,6.528,148.845
C08965=1162.769,124.312,-54.669,-178.817,6.527,148.845
C08966=1162.775,124.063,-54.649,-178.820,6.525,148.846
C08967=1162.779,123.814,-54.630,-178.823,6.524,148.846
C08968=1162.784,123.565,-54.609,-178.825,6.522,148.847
C08969=1162.789,123.316,-54.590,-178.828,6.520,148.847
C08970=1162.794,123.066,-54.570,-178.830,6.519,148.847
C08971=1162.799,122.817,-54.551,-178.834,6.518,148.848
C08972=1162.803,122.568,-54.532,-178.836,6.516,148.848
C08973=1162.808,122.319,-54.512,-178.839,6.514,148.849
C08974=1162.813,122.070,-54.493,-178.842,6.513,148.849
C08975=1162.818,121.820,-54.473,-178.844,6.511,148.850
C08976=1162.823,121.571,-54.453,-178.847,6.509,148.850
C08977=1162.827,121.323,-54.434,-178.850,6.509,148.851
C08978=1162.832,121.073,-54.415,-178.852,6.507,148.851
C08979=1162.837,120.823,-54.395,-178.855,6.505,148.851
C08980=1162.842,120.575,-54.376,-178.858,6.504,148.852
C08981=1162.847,120.325,-54.356,-178.861,6.502,148.852
C08982=1162.851,120.076,-54.337,-178.863,6.500,148.853
C08983=1162.856,119.827,-54.318,-178.866,6.499,148.853
C08984=1162.861,119.577,-54.298,-178.869,6.498,148.854
C08985=1162.866,119.328,-54.279,-178.871,6.496,148.854
C08986=1162.870,119.079,-54.260,-178.874,6.494,148.854
C08987=1162.875,118.830,-54.240,-178.877,6.493,148.855
C08988=1162.880,118.581,-54.221,-178.879,6.491,148.855
C08989=1162.885,118.332,-54.202,-178.883,6.490,148.856
C08990=1162.890,118.082,-54.183,-178.885,6.489,148.856
C08991=1162.895,117.833,-54.164,-178.887,6.487,148.857
C08992=1162.899,117.584,-54.145,-178.890,6.485,148.857
C08993=1162.904,117.334,-54.125,-178.893,6.484,148.857
C08994=1162.909,117.085,-54.106,-178.896,6.482,148.858
C08995=1162.914,116.836,-54.086,-178.899,6.481,148.858
C08996=1162.919,116.587,-54.067,-178.901,6.480,148.859
C08997=1162.923,116.338,-54.048,-178.904,6.478,148.859
C08998=1162.928,116.089,-54.030,-178.906,6.476,148.860
C08999=1162.933,115.839,-54.010,-178.910,6.475,148.860
C09000=1162.938,115.590,-53.991,-178.912,6.473,148.861
C09001=1162.942,115.341,-53.972,-178.914,6.472,148.861
C09002=1162.948,115.092,-53.953,-178.917,6.470,148.862
C09003=1162.953,114.842,-53.934,-178.920,6.469,148.862
C09004=1162.957,114.593,-53.915,-178.923,6.467,148.863
C09005=1162.962,114.344,-53.895,-178.926,6.466,148.863
C09006=1162.967,114.095,-53.877,-178.928,6.465,148.863
C09007=1162.971,113.846,-53.857,-178.931,6.463,148.864
C09008=1162.977,113.596,-53.838,-178.934,6.462,148.864
C09009=1162.981,113.347,-53.819,-178.937,6.460,148.865
C09010=1162.986,113.098,-53.800,-178.939,6.458,148.865
C09011=1162.991,112.849,-53.782,-178.941,6.457,148.866
C09012=1162.996,112.599,-53.762,-178.944,6.456,148.866
C09013=1163.001,112.351,-53.744,-178.947,6.454,148.867
C09014=1163.006,112.101,-53.725,-178.950,6.453,148.867
C09015=1163.010,111.852,-53.706,-178.953,6.451,148.867
C09016=1163.015,111.602,-53.686,-178.955,6.450,148.868
C09017=1163.020,111.353,-53.668,-178.958,6.448,148.868
C09018=1163.025,111.104,-53.649,-178.961,6.447,148.869
C09019=1163.029,110.855,-53.630,-178.963,6.445,148.869
C09020=1163.035,110.606,-53.611,-178.966,6.444,148.870
C09021=1163.039,110.356,-53.592,-178.968,6.443,148.870
C09022=1163.045,110.107,-53.574,-178.972,6.441,148.871
C09023=1163.049,109.858,-53.555,-178.974,6.440,148.871
C09024=1163.054,109.609,-53.535,-178.977,6.438,148.872
C09025=1163.059,109.360,-53.517,-178.979,6.437,148.872
C09026=1163.064,109.110,-53.498,-178.982,6.436,148.873
C09027=1163.069,108.861,-53.480,-178.985,6.434,148.873
C09028=1163.074,108.612,-53.461,-178.988,6.432,148.873
C09029=1163.078,108.362,-53.442,-178.990,6.431,148.874
C09030=1163.083,108.114,-53.424,-178.993,6.430,148.875
C09031=1163.088,107.863,-53.405,-178.996,6.428,148.875
C09032=1163.093,107.615,-53.386,-178.999,6.427,148.875
C09033=1163.098,107.365,-53.367,-179.001,6.425,148.876
C09034=1163.102,107.116,-53.348,-179.004,6.424,148.876
C09035=1163.107,106.867,-53.330,-179.007,6.423,148.877
C09036=1163.112,106.618,-53.311,-179.009,6.421,148.877
C09037=1163.117,106.349,-53.291,-179.012,6.419,148.878
C09038=1163.123,106.080,-53.271,-179.015,6.418,148.878
C09039=1163.128,105.813,-53.251,-179.018,6.416,148.879
C09040=1163.133,105.544,-53.231,-179.021,6.415,148.879
C09041=1163.138,105.294,-53.213,-179.023,6.414,148.880
C09042=1163.142,105.046,-53.194,-179.026,6.412,148.880
C09043=1163.148,104.796,-53.175,-179.029,6.411,148.881
C09044=1163.152,104.546,-53.157,-179.032,6.409,148.881
C09045=1163.157,104.298,-53.138,-179.034,6.408,148.882
C09046=1163.162,104.048,-53.120,-179.037,6.406,148.882
C09047=1163.167,103.799,-53.102,-179.040,6.405,148.883
C09048=1163.171,103.550,-53.083,-179.043,6.403,148.883
C09049=1163.177,103.301,-53.064,-179.045,6.403,148.883
C09050=1163.182,103.051,-53.046,-179.048,6.401,148.884
C09051=1163.186,102.802,-53.027,-179.051,6.399,148.885
C09052=1163.191,102.553,-53.009,-179.053,6.399,148.885
C09053=1163.197,102.303,-52.991,-179.056,6.397,148.885
C09054=1163.201,102.054,-52.973,-179.059,6.396,148.886
C09055=1163.205,101.805,-52.954,-179.062,6.394,148.886
C09056=1163.210,101.556,-52.936,-179.064,6.393,148.887
C09057=1163.216,101.306,-52.917,-179.066,6.391,148.887
C09058=1163.221,101.057,-52.899,-179.070,6.390,148.888
C09059=1163.225,100.807,-52.881,-179.072,6.389,148.888
C09060=1163.230,100.559,-52.862,-179.074,6.387,148.889
C09061=1163.235,100.310,-52.844,-179.078,6.386,148.889
C09062=1163.240,100.060,-52.826,-179.080,6.384,148.890
C09063=1163.245,99.810,-52.807,-179.083,6.383,148.890
C09064=1163.250,99.561,-52.789,-179.085,6.382,148.891
C09065=1163.255,99.312,-52.771,-179.088,6.380,148.891
C09066=1163.259,99.063,-52.752,-179.091,6.379,148.892
C09067=1163.264,98.814,-52.734,-179.093,6.378,148.892
C09068=1163.268,98.564,-52.716,-179.097,6.376,148.893
C09069=1163.274,98.315,-52.698,-179.099,6.375,148.893
C09070=1163.279,98.066,-52.680,-179.101,6.374,148.894
C09071=1163.284,97.816,-52.662,-179.104,6.372,148.894
C09072=1163.289,97.567,-52.644,-179.107,6.371,148.895
C09073=1163.294,97.318,-52.626,-179.109,6.370,148.895
C09074=1163.298,97.068,-52.607,-179.112,6.368,148.895
C09075=1163.303,96.819,-52.589,-179.115,6.367,148.896
C09076=1163.308,96.570,-52.571,-179.118,6.366,148.896
C09077=1163.313,96.321,-52.553,-179.120,6.364,148.897
C09078=1163.318,96.071,-52.535,-179.123,6.363,148.898
C09079=1163.323,95.822,-52.517,-179.126,6.362,148.898
C09080=1163.328,95.572,-52.498,-179.128,6.360,148.898
C09081=1163.333,95.323,-52.480,-179.131,6.359,148.899
C09082=1163.337,95.074,-52.462,-179.134,6.358,148.899
C09083=1163.342,94.825,-52.445,-179.136,6.356,148.900
C09084=1163.347,94.575,-52.427,-179.139,6.355,148.900
C09085=1163.352,94.326,-52.409,-179.142,6.354,148.901
C09086=1163.357,94.077,-52.391,-179.144,6.352,148.901
C09087=1163.362,93.828,-52.373,-179.147,6.351,148.902
C09088=1163.367,93.579,-52.355,-179.150,6.350,148.902
C09089=1163.371,93.329,-52.336,-179.153,6.348,148.903
C09090=1163.376,93.080,-52.318,-179.155,6.347,148.903
C09091=1163.381,92.830,-52.301,-179.158,6.346,148.904
C09092=1163.386,92.581,-52.283,-179.161,6.345,148.904
C09093=1163.391,92.331,-52.265,-179.163,6.343,148.905
C09094=1163.396,92.082,-52.247,-179.166,6.342,148.905
C09095=1163.401,91.833,-52.229,-179.169,6.341,148.906
C09096=1163.406,91.584,-52.211,-179.171,6.339,148.906
C09097=1163.411,91.335,-52.193,-179.174,6.338,148.907
C09098=1163.415,91.085,-52.176,-179.177,6.337,148.907
C09099=1163.420,90.836,-52.158,-179.179,6.336,148.908
C09100=1163.425,90.587,-52.141,-179.182,6.334,148.908
C09101=1163.430,90.338,-52.123,-179.185,6.333,148.909
C09102=1163.435,90.088,-52.105,-179.187,6.332,148.909
C09103=1163.440,89.839,-52.087,-179.190,6.331,148.910
C09104=1163.445,89.590,-52.069,-179.193,6.329,148.910
C09105=1163.449,89.340,-52.051,-179.195,6.328,148.911
C09106=1163.455,89.090,-52.034,-179.198,6.327,148.911
C09107=1163.460,88.841,-52.016,-179.201,6.325,148.912
C09108=1163.464,88.592,-51.998,-179.203,6.324,148.912
C09109=1163.469,88.343,-51.980,-179.206,6.323,148.913
C09110=1163.474,88.093,-51.963,-179.208,6.322,148.913
C09111=1163.479,87.844,-51.945,-179.211,6.320,148.914
C09112=1163.484,87.595,-51.927,-179.214,6.319,148.914
C09113=1163.489,87.345,-51.910,-179.217,6.318,148.915
C09114=1163.493,87.096,-51.892,-179.219,6.316,148.915
C09115=1163.498,86.846,-51.875,-179.222,6.316,148.916
C09116=1163.504,86.598,-51.858,-179.225,6.314,148.916
C09117=1163.509,86.348,-51.840,-179.227,6.312,148.917
C09118=1163.514,86.099,-51.822,-179.230,6.312,148.917
C09119=1163.518,85.850,-51.805,-179.233,6.310,148.918
C09120=1163.523,85.600,-51.788,-179.236,6.309,148.918
C09121=1163.528,85.351,-51.770,-179.238,6.308,148.919
C09122=1163.533,85.102,-51.752,-179.241,6.306,148.919
C09123=1163.538,84.852,-51.735,-179.243,6.306,148.920
C09124=1163.542,84.603,-51.717,-179.246,6.304,148.920
C09125=1163.548,84.353,-51.700,-179.249,6.302,148.921
C09126=1163.553,84.104,-51.682,-179.252,6.302,148.921
C09127=1163.557,83.855,-51.665,-179.254,6.300,148.922
C09128=1163.562,83.605,-51.647,-179.256,6.299,148.922
C09129=1163.567,83.356,-51.630,-179.260,6.298,148.923
C09130=1163.572,83.106,-51.612,-179.262,6.296,148.923
C09131=1163.577,82.857,-51.595,-179.265,6.296,148.924
C09132=1163.582,82.608,-51.577,-179.268,6.294,148.924
C09133=1163.587,82.359,-51.560,-179.270,6.293,148.925
C09134=1163.592,82.110,-51.543,-179.273,6.292,148.925
C09135=1163.597,81.860,-51.526,-179.275,6.291,148.926
C09136=1163.602,81.610,-51.509,-179.278,6.289,148.926
C09137=1163.606,81.361,-51.491,-179.281,6.288,148.927
C09138=1163.611,81.112,-51.474,-179.283,6.287,148.927
C09139=1163.616,80.862,-51.456,-179.286,6.286,148.928
C09140=1163.621,80.613,-51.439,-179.289,6.285,148.928
C09141=1163.627,80.345,-51.421,-179.291,6.283,148.929
C09142=1163.632,80.076,-51.401,-179.295,6.282,148.929
C09143=1163.636,79.808,-51.383,-179.298,6.280,148.930
C09144=1163.642,79.540,-51.365,-179.300,6.280,148.931
C09145=1163.648,79.290,-51.348,-179.303,6.278,148.931
C09146=1163.652,79.041,-51.330,-179.305,6.277,148.932
C09147=1163.657,78.791,-51.313,-179.308,6.276,148.932
C09148=1163.662,78.541,-51.296,-179.311,6.274,148.933
C09149=1163.667,78.293,-51.279,-179.313,6.273,148.933
